C05440=1057.096,54.680,-74.753,171.430,30.537,155.701
C05441=1057.102,54.929,-74.770,171.432,30.540,155.701
C05442=1057.108,55.179,-74.788,171.434,30.542,155.702
C05443=1057.114,55.428,-74.804,171.435,30.544,155.702
C05444=1057.121,55.677,-74.821,171.437,30.547,155.703
C05445=1057.126,55.927,-74.838,171.438,30.549,155.703
C05446=1057.133,56.176,-74.855,171.439,30.552,155.703
C05447=1057.139,56.426,-74.873,171.441,30.554,155.704
C05448=1057.145,56.675,-74.889,171.443,30.557,155.704
C05449=1057.152,56.924,-74.907,171.445,30.559,155.704
C05450=1057.157,57.173,-74.924,171.445,30.561,155.705
C05451=1057.163,57.422,-74.941,171.447,30.563,155.705
C05452=1057.170,57.672,-74.958,171.449,30.566,155.705
C05453=1057.175,57.921,-74.975,171.451,30.568,155.706
C05454=1057.182,58.171,-74.993,171.452,30.571,155.706
C05455=1057.187,58.420,-75.009,171.453,30.573,155.706
C05456=1057.194,58.670,-75.027,171.455,30.576,155.707
C05457=1057.201,58.918,-75.044,171.456,30.578,155.707
C05458=1057.207,59.168,-75.062,171.458,30.580,155.708
C05459=1057.213,59.418,-75.078,171.460,30.583,155.708
C05460=1057.219,59.667,-75.096,171.461,30.585,155.708
C05461=1057.225,59.916,-75.113,171.462,30.588,155.709
C05462=1057.232,60.165,-75.130,171.464,30.590,155.709
C05463=1057.237,60.415,-75.147,171.466,30.593,155.709
C05464=1057.243,60.664,-75.164,171.467,30.594,155.710
C05465=1057.249,60.914,-75.182,171.468,30.597,155.710
C05466=1057.256,61.162,-75.199,171.470,30.599,155.710
C05467=1057.263,61.412,-75.216,171.472,30.602,155.711
C05468=1057.269,61.697,-75.236,171.474,30.605,155.711
C05469=1057.277,61.982,-75.256,171.476,30.607,155.712
C05470=1057.283,62.267,-75.276,171.477,30.610,155.712
C05471=1057.291,62.551,-75.295,171.479,30.613,155.712
C05472=1057.297,62.801,-75.313,171.480,30.615,155.713
C05473=1057.303,63.051,-75.329,171.482,30.618,155.713
C05474=1057.309,63.300,-75.347,171.484,30.620,155.713
C05475=1057.316,63.550,-75.365,171.485,30.622,155.714
C05476=1057.321,63.799,-75.382,171.486,30.624,155.714
C05477=1057.328,64.048,-75.400,171.488,30.627,155.714
C05478=1057.334,64.297,-75.417,171.490,30.629,155.715
C05479=1057.341,64.547,-75.435,171.491,30.632,155.715
C05480=1057.346,64.796,-75.452,171.493,30.634,155.715
C05481=1057.352,65.045,-75.470,171.494,30.636,155.716
C05482=1057.358,65.294,-75.487,171.496,30.639,155.716
C05483=1057.365,65.544,-75.505,171.497,30.641,155.717
C05484=1057.370,65.793,-75.522,171.499,30.644,155.717
C05485=1057.377,66.042,-75.540,171.500,30.647,155.717
C05486=1057.382,66.291,-75.557,171.501,30.649,155.718
C05487=1057.389,66.541,-75.575,171.503,30.651,155.718
C05488=1057.395,66.790,-75.592,171.505,30.653,155.718
C05489=1057.401,67.040,-75.610,171.507,30.656,155.719
C05490=1057.406,67.289,-75.628,171.508,30.659,155.719
C05491=1057.413,67.538,-75.645,171.509,30.661,155.720
C05492=1057.419,67.788,-75.663,171.511,30.663,155.720
C05493=1057.425,68.037,-75.681,171.512,30.666,155.720
C05494=1057.431,68.287,-75.699,171.514,30.668,155.721
C05495=1057.437,68.535,-75.716,171.516,30.671,155.721
C05496=1057.443,68.785,-75.733,171.517,30.673,155.721
C05497=1057.449,69.034,-75.751,171.518,30.675,155.722
C05498=1057.455,69.284,-75.769,171.520,30.678,155.722
C05499=1057.461,69.533,-75.786,171.522,30.680,155.722
C05500=1057.467,69.782,-75.804,171.524,30.683,155.723
C05501=1057.474,70.031,-75.823,171.524,30.685,155.723
C05502=1057.479,70.280,-75.840,171.526,30.688,155.724
C05503=1057.486,70.530,-75.858,171.528,30.690,155.724
C05504=1057.492,70.779,-75.875,171.529,30.693,155.724
C05505=1057.498,71.029,-75.893,171.531,30.695,155.725
C05506=1057.503,71.278,-75.911,171.532,30.698,155.725
C05507=1057.510,71.527,-75.928,171.534,30.700,155.726
C05508=1057.516,71.777,-75.947,171.535,30.702,155.726
C05509=1057.522,72.026,-75.965,171.537,30.705,155.726
C05510=1057.528,72.275,-75.982,171.539,30.708,155.727
C05511=1057.534,72.524,-76.000,171.540,30.710,155.727
C05512=1057.540,72.774,-76.017,171.541,30.712,155.727
C05513=1057.546,73.023,-76.036,171.543,30.715,155.728
C05514=1057.552,73.272,-76.054,171.545,30.717,155.728
C05515=1057.558,73.522,-76.072,171.546,30.720,155.728
C05516=1057.564,73.771,-76.089,171.548,30.722,155.729
C05517=1057.570,74.020,-76.108,171.549,30.725,155.729
C05518=1057.576,74.270,-76.126,171.550,30.727,155.730
C05519=1057.582,74.519,-76.143,171.552,30.730,155.730
C05520=1057.589,74.768,-76.161,171.554,30.732,155.730
C05521=1057.594,75.017,-76.179,171.556,30.735,155.731
C05522=1057.600,75.266,-76.197,171.556,30.737,155.731
C05523=1057.607,75.516,-76.215,171.558,30.739,155.731
C05524=1057.612,75.764,-76.233,171.560,30.742,155.732
C05525=1057.619,76.014,-76.251,171.561,30.744,155.732
C05526=1057.625,76.264,-76.269,171.563,30.747,155.733
C05527=1057.630,76.512,-76.287,171.564,30.749,155.733
C05528=1057.637,76.762,-76.305,171.566,30.752,155.733
C05529=1057.643,77.012,-76.323,171.567,30.754,155.734
C05530=1057.649,77.260,-76.341,171.569,30.757,155.734
C05531=1057.655,77.510,-76.359,171.571,30.759,155.734
C05532=1057.662,77.795,-76.380,171.572,30.762,155.735
C05533=1057.669,78.080,-76.400,171.574,30.765,155.735
C05534=1057.676,78.364,-76.421,171.576,30.767,155.736
C05535=1057.683,78.649,-76.442,171.578,30.771,155.736
C05536=1057.689,78.899,-76.460,171.579,30.773,155.737
C05537=1057.695,79.147,-76.478,171.580,30.775,155.737
C05538=1057.700,79.397,-76.497,171.582,30.778,155.737
C05539=1057.706,79.647,-76.515,171.584,30.781,155.738
C05540=1057.712,79.896,-76.533,171.585,30.783,155.738
C05541=1057.718,80.145,-76.551,171.587,30.785,155.738
C05542=1057.725,80.394,-76.570,171.588,30.788,155.739
C05543=1057.730,80.643,-76.587,171.589,30.791,155.739
C05544=1057.736,80.893,-76.606,171.591,30.793,155.740
C05545=1057.742,81.143,-76.624,171.593,30.795,155.740
C05546=1057.748,81.391,-76.643,171.595,30.798,155.740
C05547=1057.754,81.641,-76.661,171.596,30.801,155.741
C05548=1057.760,81.890,-76.679,171.597,30.803,155.741
C05549=1057.766,82.139,-76.697,171.599,30.805,155.742
C05550=1057.772,82.388,-76.716,171.601,30.808,155.742
C05551=1057.778,82.638,-76.735,171.602,30.811,155.742
C05552=1057.784,82.887,-76.753,171.604,30.813,155.743
C05553=1057.790,83.136,-76.771,171.605,30.815,155.743
C05554=1057.796,83.385,-76.789,171.606,30.818,155.744
C05555=1057.802,83.635,-76.807,171.608,30.821,155.744
C05556=1057.808,83.885,-76.826,171.610,30.823,155.744
C05557=1057.814,84.133,-76.844,171.612,30.825,155.745
C05558=1057.820,84.382,-76.863,171.613,30.828,155.745
C05559=1057.826,84.632,-76.881,171.614,30.830,155.745
C05560=1057.833,84.881,-76.899,171.616,30.833,155.746
C05561=1057.837,85.130,-76.918,171.618,30.835,155.746
C05562=1057.844,85.379,-76.936,171.619,30.838,155.747
C05563=1057.850,85.629,-76.955,171.621,30.840,155.747
C05564=1057.856,85.878,-76.973,171.622,30.843,155.747
C05565=1057.862,86.127,-76.991,171.623,30.845,155.748
C05566=1057.868,86.376,-77.010,171.625,30.847,155.748
C05567=1057.874,86.626,-77.028,171.627,30.850,155.748
C05568=1057.880,86.875,-77.047,171.629,30.853,155.749
C05569=1057.887,87.124,-77.066,171.630,30.855,155.749
C05570=1057.892,87.373,-77.083,171.631,30.857,155.750
C05571=1057.898,87.623,-77.102,171.633,30.860,155.750
C05572=1057.905,87.872,-77.121,171.635,30.863,155.750
C05573=1057.911,88.121,-77.140,171.636,30.865,155.751
C05574=1057.917,88.371,-77.158,171.638,30.867,155.751
C05575=1057.923,88.619,-77.176,171.639,30.870,155.752
C05576=1057.929,88.868,-77.195,171.641,30.872,155.752
C05577=1057.935,89.118,-77.214,171.642,30.875,155.752
C05578=1057.941,89.367,-77.232,171.644,30.877,155.753
C05579=1057.948,89.616,-77.250,171.646,30.880,155.753
C05580=1057.953,89.866,-77.270,171.648,30.882,155.753
C05581=1057.960,90.115,-77.288,171.648,30.885,155.754
C05582=1057.965,90.364,-77.306,171.650,30.887,155.754
C05583=1057.972,90.613,-77.325,171.652,30.890,155.754
C05584=1057.977,90.863,-77.344,171.654,30.892,155.755
C05585=1057.984,91.112,-77.362,171.655,30.895,155.755
C05586=1057.989,91.361,-77.382,171.656,30.897,155.756
C05587=1057.996,91.610,-77.400,171.658,30.900,155.756
C05588=1058.001,91.860,-77.418,171.659,30.902,155.756
C05589=1058.007,92.109,-77.437,171.661,30.905,155.757
C05590=1058.013,92.358,-77.456,171.663,30.907,155.757
C05591=1058.019,92.607,-77.475,171.665,30.910,155.758
C05592=1058.025,92.857,-77.494,171.665,30.912,155.758
C05593=1058.031,93.106,-77.513,171.667,30.915,155.758
C05594=1058.036,93.355,-77.532,171.669,30.917,155.759
C05595=1058.043,93.604,-77.550,171.671,30.920,155.759
C05596=1058.049,93.889,-77.572,171.673,30.923,155.760
C05597=1058.057,94.174,-77.593,171.674,30.926,155.760
C05598=1058.063,94.458,-77.615,171.676,30.929,155.761
C05599=1058.070,94.743,-77.637,171.678,30.931,155.761
C05600=1058.076,94.992,-77.655,171.679,30.934,155.761
C05601=1058.082,95.242,-77.675,171.681,30.937,155.762
C05602=1058.089,95.491,-77.693,171.682,30.939,155.762
C05603=1058.094,95.740,-77.712,171.684,30.941,155.763
C05604=1058.101,95.990,-77.731,171.685,30.944,155.763
C05605=1058.106,96.239,-77.750,171.687,30.947,155.763
C05606=1058.112,96.487,-77.769,171.689,30.949,155.764
C05607=1058.118,96.737,-77.788,171.691,30.951,155.764
C05608=1058.124,96.986,-77.806,171.691,30.954,155.764
C05609=1058.130,97.235,-77.826,171.693,30.957,155.765
C05610=1058.136,97.484,-77.844,171.695,30.959,155.765
C05611=1058.142,97.734,-77.864,171.697,30.961,155.766
C05612=1058.148,97.983,-77.883,171.698,30.964,155.766
C05613=1058.154,98.232,-77.902,171.700,30.967,155.766
C05614=1058.160,98.482,-77.921,171.701,30.969,155.767
C05615=1058.166,98.731,-77.939,171.703,30.971,155.767
C05616=1058.172,98.980,-77.959,171.704,30.974,155.768
C05617=1058.178,99.230,-77.977,171.706,30.977,155.768
C05618=1058.184,99.478,-77.997,171.708,30.979,155.768
C05619=1058.191,99.728,-78.016,171.710,30.981,155.769
C05620=1058.197,99.977,-78.035,171.710,30.984,155.769
C05621=1058.203,100.226,-78.054,171.712,30.987,155.770
C05622=1058.209,100.476,-78.073,171.714,30.989,155.770
C05623=1058.215,100.725,-78.092,171.716,30.991,155.770
C05624=1058.221,100.974,-78.111,171.718,30.994,155.771
C05625=1058.227,101.223,-78.131,171.718,30.997,155.771
C05626=1058.232,101.472,-78.150,171.720,30.999,155.772
C05627=1058.239,101.721,-78.169,171.722,31.002,155.772
C05628=1058.245,101.971,-78.188,171.724,31.004,155.772
C05629=1058.250,102.220,-78.207,171.725,31.006,155.773
C05630=1058.256,102.468,-78.227,171.727,31.009,155.773
C05631=1058.262,102.718,-78.246,171.728,31.012,155.773
C05632=1058.268,102.967,-78.265,171.730,31.015,155.774
C05633=1058.273,103.216,-78.284,171.731,31.017,155.774
C05634=1058.279,103.465,-78.304,171.733,31.019,155.775
C05635=1058.285,103.715,-78.323,171.735,31.022,155.775
C05636=1058.292,103.964,-78.342,171.737,31.024,155.775
C05637=1058.298,104.213,-78.362,171.737,31.027,155.776
C05638=1058.303,104.462,-78.381,171.739,31.030,155.776
C05639=1058.309,104.711,-78.400,171.741,31.032,155.777
C05640=1058.315,104.961,-78.419,171.743,31.034,155.777
C05641=1058.321,105.209,-78.439,171.744,31.037,155.777
C05642=1058.327,105.459,-78.458,171.746,31.040,155.778
C05643=1058.333,105.708,-78.477,171.747,31.042,155.778
C05644=1058.339,105.957,-78.497,171.749,31.045,155.779
C05645=1058.345,106.206,-78.516,171.751,31.048,155.779
C05646=1058.351,106.456,-78.535,171.752,31.050,155.779
C05647=1058.357,106.704,-78.555,171.754,31.052,155.780
C05648=1058.363,106.955,-78.575,171.756,31.055,155.780
C05649=1058.369,107.203,-78.595,171.757,31.058,155.781
C05650=1058.376,107.452,-78.613,171.758,31.060,155.781
C05651=1058.381,107.702,-78.633,171.760,31.062,155.781
C05652=1058.387,107.951,-78.653,171.762,31.065,155.782
C05653=1058.393,108.200,-78.672,171.764,31.068,155.782
C05654=1058.399,108.449,-78.692,171.765,31.070,155.783
C05655=1058.405,108.698,-78.711,171.766,31.073,155.783
C05656=1058.411,108.947,-78.730,171.768,31.075,155.783
C05657=1058.417,109.196,-78.750,171.770,31.077,155.784
C05658=1058.423,109.446,-78.769,171.772,31.080,155.784
C05659=1058.429,109.695,-78.789,171.773,31.083,155.785
C05660=1058.436,109.980,-78.811,171.775,31.085,155.785
C05661=1058.443,110.264,-78.834,171.777,31.088,155.785
C05662=1058.450,110.550,-78.856,171.779,31.091,155.786
C05663=1058.457,110.835,-78.878,171.781,31.094,155.786
C05664=1058.463,111.083,-78.898,171.782,31.097,155.787
C05665=1058.469,111.333,-78.917,171.784,31.099,155.787
C05666=1058.475,111.582,-78.937,171.785,31.102,155.788
C05667=1058.481,111.830,-78.957,171.787,31.104,155.788
C05668=1058.486,112.080,-78.976,171.789,31.107,155.788
C05669=1058.492,112.329,-78.996,171.790,31.109,155.789
C05670=1058.498,112.578,-79.015,171.792,31.112,155.789
C05671=1058.505,112.828,-79.036,171.794,31.115,155.790
C05672=1058.510,113.077,-79.055,171.795,31.117,155.790
C05673=1058.516,113.326,-79.075,171.797,31.119,155.790
C05674=1058.522,113.575,-79.095,171.798,31.122,155.791
C05675=1058.528,113.824,-79.114,171.800,31.124,155.791
C05676=1058.534,114.073,-79.134,171.802,31.127,155.791
C05677=1058.540,114.322,-79.154,171.804,31.130,155.792
C05678=1058.546,114.571,-79.173,171.805,31.132,155.792
C05679=1058.551,114.821,-79.194,171.806,31.135,155.793
C05680=1058.557,115.070,-79.214,171.808,31.138,155.793
C05681=1058.563,115.319,-79.233,171.810,31.140,155.794
C05682=1058.569,115.568,-79.253,171.812,31.143,155.794
C05683=1058.575,115.817,-79.273,171.814,31.146,155.794
C05684=1058.580,116.067,-79.293,171.814,31.148,155.795
C05685=1058.586,116.315,-79.313,171.816,31.151,155.795
C05686=1058.592,116.564,-79.333,171.818,31.153,155.796
C05687=1058.598,116.813,-79.353,171.820,31.156,155.796
C05688=1058.604,117.064,-79.373,171.822,31.158,155.796
C05689=1058.610,117.312,-79.393,171.823,31.161,155.797
C05690=1058.616,117.561,-79.413,171.824,31.163,155.797
C05691=1058.622,117.810,-79.433,171.826,31.166,155.798
C05692=1058.627,118.059,-79.452,171.828,31.169,155.798
C05693=1058.633,118.309,-79.473,171.830,31.171,155.798
C05694=1058.639,118.558,-79.493,171.831,31.174,155.799
C05695=1058.645,118.807,-79.513,171.833,31.177,155.799
C05696=1058.651,119.056,-79.533,171.834,31.179,155.800
C05697=1058.656,119.305,-79.553,171.836,31.182,155.800
C05698=1058.662,119.554,-79.573,171.838,31.185,155.801
C05699=1058.668,119.803,-79.593,171.839,31.187,155.801
C05700=1058.675,120.053,-79.613,171.841,31.190,155.801
C05701=1058.680,120.302,-79.634,171.843,31.192,155.802
C05702=1058.686,120.551,-79.654,171.844,31.194,155.802
C05703=1058.692,120.799,-79.674,171.846,31.197,155.803
C05704=1058.698,121.049,-79.693,171.847,31.200,155.803
C05705=1058.703,121.299,-79.714,171.849,31.202,155.803
C05706=1058.709,121.547,-79.734,171.851,31.205,155.804
C05707=1058.715,121.796,-79.754,171.853,31.208,155.804
C05708=1058.721,122.045,-79.774,171.854,31.210,155.805
C05709=1058.727,122.295,-79.795,171.856,31.213,155.805
C05710=1058.733,122.544,-79.815,171.857,31.215,155.805
C05711=1058.739,122.792,-79.835,171.859,31.218,155.806
C05712=1058.745,123.042,-79.855,171.861,31.220,155.806
C05713=1058.751,123.291,-79.876,171.863,31.223,155.807
C05714=1058.757,123.540,-79.895,171.865,31.225,155.807
C05715=1058.763,123.789,-79.915,171.866,31.228,155.807
C05716=1058.769,124.039,-79.936,171.867,31.231,155.808
C05717=1058.775,124.287,-79.956,171.869,31.233,155.808
C05718=1058.781,124.536,-79.976,171.871,31.236,155.809
C05719=1058.786,124.785,-79.997,171.873,31.239,155.809
C05720=1058.793,125.035,-80.017,171.875,31.241,155.810
C05721=1058.799,125.284,-80.037,171.876,31.243,155.810
C05722=1058.804,125.533,-80.058,171.877,31.246,155.810
C05723=1058.811,125.782,-80.078,171.879,31.248,155.811
C05724=1058.817,126.067,-80.101,171.881,31.252,155.811
C05725=1058.824,126.351,-80.124,171.884,31.255,155.812
C05726=1058.831,126.636,-80.147,171.886,31.257,155.812
C05727=1058.838,126.921,-80.171,171.887,31.260,155.813
C05728=1058.844,127.170,-80.191,171.889,31.263,155.813
C05729=1058.850,127.419,-80.211,171.890,31.266,155.813
C05730=1058.855,127.669,-80.232,171.892,31.268,155.814
C05731=1058.862,127.917,-80.252,171.894,31.270,155.814
C05732=1058.868,128.167,-80.273,171.896,31.273,155.815
C05733=1058.874,128.415,-80.293,171.897,31.276,155.815
C05734=1058.880,128.664,-80.313,171.899,31.278,155.815
C05735=1058.886,128.914,-80.334,171.901,31.281,155.816
C05736=1058.891,129.163,-80.354,171.903,31.284,155.816
C05737=1058.897,129.412,-80.374,171.904,31.285,155.817
C05738=1058.904,129.661,-80.395,171.906,31.288,155.817
C05739=1058.910,129.910,-80.416,171.908,31.291,155.817
C05740=1058.916,130.159,-80.436,171.909,31.293,155.818
C05741=1058.922,130.408,-80.456,171.911,31.296,155.818
C05742=1058.928,130.658,-80.477,171.913,31.299,155.819
C05743=1058.934,130.906,-80.498,171.915,31.301,155.819
C05744=1058.940,131.155,-80.518,171.917,31.303,155.819
C05745=1058.946,131.405,-80.538,171.918,31.306,155.820
C05746=1058.952,131.654,-80.558,171.920,31.309,155.820
C05747=1058.958,131.903,-80.580,171.921,31.311,155.821
C05748=1058.964,132.152,-80.600,171.923,31.314,155.821
C05749=1058.970,132.401,-80.621,171.925,31.317,155.821
C05750=1058.976,132.650,-80.641,171.927,31.319,155.822
C05751=1058.982,132.899,-80.662,171.929,31.322,155.822
C05752=1058.988,133.149,-80.683,171.930,31.324,155.823
C05753=1058.994,133.398,-80.703,171.931,31.327,155.823
C05754=1058.999,133.646,-80.724,171.933,31.330,155.824
C05755=1059.005,133.896,-80.745,171.935,31.332,155.824
C05756=1059.011,134.144,-80.766,171.937,31.335,155.824
C05757=1059.017,134.394,-80.787,171.939,31.338,155.825
C05758=1059.023,134.643,-80.807,171.941,31.340,155.825
C05759=1059.029,134.891,-80.828,171.943,31.343,155.826
C05760=1059.035,135.141,-80.849,171.944,31.346,155.826
C05761=1059.041,135.390,-80.869,171.945,31.348,155.826
C05762=1059.047,135.639,-80.891,171.947,31.351,155.827
C05763=1059.052,135.888,-80.911,171.949,31.353,155.827
C05764=1059.059,136.137,-80.932,171.951,31.356,155.828
C05765=1059.064,136.386,-80.953,171.953,31.358,155.828
C05766=1059.070,136.635,-80.974,171.954,31.361,155.828
C05767=1059.076,136.884,-80.994,171.956,31.363,155.829
C05768=1059.082,137.133,-81.016,171.958,31.366,155.829
C05769=1059.088,137.382,-81.036,171.960,31.369,155.830
C05770=1059.094,137.631,-81.057,171.961,31.371,155.830
C05771=1059.100,137.881,-81.078,171.963,31.374,155.831
C05772=1059.105,138.129,-81.099,171.965,31.376,155.831
C05773=1059.112,138.379,-81.120,171.966,31.379,155.831
C05774=1059.118,138.627,-81.141,171.968,31.382,155.832
C05775=1059.123,138.877,-81.162,171.970,31.384,155.832
C05776=1059.129,139.125,-81.183,171.972,31.387,155.833
C05777=1059.136,139.375,-81.203,171.974,31.390,155.833
C05778=1059.141,139.623,-81.225,171.976,31.392,155.833
C05779=1059.147,139.873,-81.246,171.978,31.395,155.834
C05780=1059.153,140.121,-81.266,171.979,31.398,155.834
C05781=1059.160,140.371,-81.288,171.980,31.400,155.835
C05782=1059.165,140.620,-81.309,171.982,31.403,155.835
C05783=1059.171,140.869,-81.330,171.984,31.405,155.836
C05784=1059.176,141.118,-81.351,171.986,31.408,155.836
C05785=1059.182,141.367,-81.372,171.988,31.411,155.836
C05786=1059.188,141.616,-81.394,171.990,31.413,155.837
C05787=1059.194,141.866,-81.415,171.991,31.416,155.837
C05788=1059.200,142.150,-81.439,171.993,31.419,155.838
C05789=1059.208,142.434,-81.463,171.995,31.422,155.838
C05790=1059.215,142.719,-81.487,171.997,31.425,155.839
C05791=1059.221,143.004,-81.511,172.000,31.428,155.839
C05792=1059.226,143.253,-81.532,172.002,31.431,155.840
C05793=1059.233,143.502,-81.554,172.003,31.434,155.840
C05794=1059.239,143.750,-81.575,172.004,31.436,155.841
C05795=1059.245,144.000,-81.596,172.006,31.439,155.841
C05796=1059.250,144.248,-81.617,172.008,31.441,155.841
C05797=1059.256,144.498,-81.639,172.010,31.444,155.842
C05798=1059.262,144.746,-81.660,172.012,31.447,155.842
C05799=1059.268,144.996,-81.681,172.014,31.449,155.843
C05800=1059.274,145.233,-81.702,172.015,31.452,155.843
C05801=1059.279,145.470,-81.721,172.017,31.455,155.843
C05802=1059.285,145.707,-81.742,172.019,31.457,155.844
C05803=1059.290,145.944,-81.762,172.021,31.459,155.844
C05804=1059.296,146.181,-81.783,172.022,31.462,155.845
C05805=1059.302,146.418,-81.802,172.024,31.464,155.845
C05806=1059.308,146.655,-81.823,172.026,31.467,155.845
C05807=1059.313,146.892,-81.843,172.027,31.470,155.846
C05808=1059.319,147.141,-81.865,172.029,31.472,155.846
C05809=1059.325,147.391,-81.886,172.031,31.475,155.847
C05810=1059.331,147.639,-81.907,172.033,31.478,155.847
C05811=1059.337,147.888,-81.929,172.035,31.480,155.848
C05812=1059.342,148.137,-81.950,172.037,31.483,155.848
C05813=1059.348,148.386,-81.972,172.039,31.485,155.848
C05814=1059.355,148.635,-81.994,172.040,31.488,155.849
C05815=1059.360,148.884,-82.015,172.042,31.491,155.849
C05816=1059.366,149.134,-82.036,172.044,31.493,155.850
C05817=1059.372,149.382,-82.057,172.045,31.496,155.850
C05818=1059.378,149.631,-82.079,172.047,31.498,155.851
C05819=1059.384,149.881,-82.100,172.049,31.501,155.851
C05820=1059.390,150.129,-82.122,172.051,31.504,155.851
C05821=1059.396,150.378,-82.143,172.052,31.506,155.852
C05822=1059.401,150.628,-82.166,172.054,31.510,155.852
C05823=1059.407,150.876,-82.187,172.056,31.512,155.853
C05824=1059.413,151.125,-82.208,172.058,31.515,155.853
C05825=1059.419,151.375,-82.230,172.060,31.517,155.854
C05826=1059.425,151.623,-82.251,172.062,31.520,155.854
C05827=1059.431,151.872,-82.273,172.064,31.523,155.854
C05828=1059.436,152.122,-82.295,172.065,31.525,155.855
C05829=1059.442,152.370,-82.317,172.067,31.528,155.855
C05830=1059.448,152.619,-82.339,172.069,31.531,155.856
C05831=1059.454,152.868,-82.360,172.071,31.533,155.856
C05832=1059.460,153.117,-82.382,172.073,31.536,155.857
C05833=1059.466,153.366,-82.403,172.075,31.539,155.857
C05834=1059.471,153.615,-82.426,172.077,31.542,155.857
C05835=1059.477,153.864,-82.447,172.078,31.544,155.858
C05836=1059.483,154.113,-82.468,172.080,31.547,155.858
C05837=1059.489,154.362,-82.490,172.082,31.550,155.859
C05838=1059.496,154.612,-82.512,172.084,31.552,155.859
C05839=1059.501,154.860,-82.534,172.086,31.555,155.860
C05840=1059.507,155.109,-82.556,172.088,31.558,155.860
C05841=1059.513,155.358,-82.578,172.090,31.560,155.860
C05842=1059.519,155.607,-82.599,172.092,31.563,155.861
C05843=1059.524,155.856,-82.621,172.093,31.566,155.861
C05844=1059.530,156.105,-82.643,172.095,31.569,155.862
C05845=1059.537,156.354,-82.665,172.097,31.571,155.862
C05846=1059.541,156.603,-82.687,172.099,31.574,155.863
C05847=1059.548,156.852,-82.709,172.101,31.576,155.863
C05848=1059.554,157.101,-82.730,172.103,31.580,155.864
C05849=1059.560,157.350,-82.753,172.105,31.582,155.864
C05850=1059.565,157.599,-82.774,172.106,31.585,155.864
C05851=1059.571,157.848,-82.796,172.108,31.588,155.865
C05852=1059.579,158.156,-82.824,172.111,31.591,155.865
C05853=1059.586,158.464,-82.851,172.113,31.594,155.866
C05854=1059.593,158.772,-82.877,172.116,31.597,155.866
C05855=1059.600,159.081,-82.905,172.118,31.601,155.867
C05856=1059.606,159.330,-82.927,172.119,31.604,155.868
C05857=1059.613,159.579,-82.949,172.121,31.607,155.868
C05858=1059.617,159.828,-82.971,172.123,31.609,155.868
C05859=1059.624,160.076,-82.993,172.125,31.612,155.869
C05860=1059.630,160.325,-83.015,172.127,31.614,155.869
C05861=1059.636,160.574,-83.038,172.129,31.617,155.870
C05862=1059.642,160.824,-83.060,172.131,31.620,155.870
C05863=1059.647,161.073,-83.082,172.133,31.623,155.871
C05864=1059.653,161.321,-83.104,172.134,31.625,155.871
C05865=1059.659,161.570,-83.126,172.136,31.628,155.871
C05866=1059.664,161.819,-83.149,172.138,31.631,155.872
C05867=1059.670,162.068,-83.170,172.140,31.634,155.872
C05868=1059.676,162.317,-83.193,172.142,31.637,155.873
C05869=1059.681,162.566,-83.215,172.144,31.640,155.873
C05870=1059.688,162.815,-83.238,172.146,31.642,155.874
C05871=1059.693,163.064,-83.260,172.147,31.645,155.874
C05872=1059.698,163.313,-83.283,172.150,31.648,155.875
C05873=1059.704,163.562,-83.304,172.152,31.651,155.875
C05874=1059.710,163.811,-83.327,172.154,31.654,155.876
C05875=1059.715,164.060,-83.349,172.156,31.657,155.876
C05876=1059.721,164.308,-83.372,172.158,31.659,155.877
C05877=1059.727,164.557,-83.394,172.160,31.662,155.877
C05878=1059.732,164.806,-83.416,172.162,31.665,155.877
C05879=1059.738,165.055,-83.439,172.163,31.668,155.878
C05880=1059.744,165.305,-83.461,172.165,31.670,155.878
C05881=1059.750,165.553,-83.484,172.167,31.674,155.879
C05882=1059.755,165.802,-83.507,172.169,31.676,155.879
C05883=1059.761,166.051,-83.529,172.171,31.679,155.880
C05884=1059.767,166.300,-83.551,172.173,31.682,155.880
C05885=1059.773,166.549,-83.573,172.175,31.685,155.881
C05886=1059.778,166.798,-83.596,172.176,31.687,155.881
C05887=1059.785,167.047,-83.619,172.178,31.690,155.882
C05888=1059.790,167.296,-83.641,172.180,31.693,155.882
C05889=1059.795,167.544,-83.664,172.182,31.696,155.883
C05890=1059.801,167.793,-83.686,172.184,31.699,155.883
C05891=1059.808,168.042,-83.709,172.187,31.702,155.883
C05892=1059.813,168.291,-83.731,172.189,31.704,155.884
C05893=1059.819,168.540,-83.754,172.191,31.707,155.884
C05894=1059.824,168.789,-83.777,172.192,31.710,155.885
C05895=1059.831,169.038,-83.799,172.194,31.713,155.885
C05896=1059.836,169.287,-83.822,172.196,31.716,155.886
C05897=1059.841,169.536,-83.844,172.198,31.719,155.886
C05898=1059.847,169.784,-83.867,172.200,31.721,155.887
C05899=1059.853,170.033,-83.890,172.202,31.724,155.887
C05900=1059.859,170.283,-83.912,172.204,31.727,155.888
C05901=1059.865,170.531,-83.935,172.206,31.730,155.888
C05902=1059.871,170.780,-83.958,172.207,31.733,155.889
C05903=1059.876,171.029,-83.980,172.210,31.735,155.889
C05904=1059.883,171.278,-84.003,172.212,31.738,155.889
C05905=1059.888,171.527,-84.026,172.214,31.741,155.890
C05906=1059.894,171.776,-84.048,172.216,31.744,155.890
C05907=1059.900,172.025,-84.071,172.218,31.747,155.891
C05908=1059.905,172.274,-84.094,172.220,31.750,155.891
C05909=1059.912,172.523,-84.116,172.222,31.752,155.892
C05910=1059.918,172.772,-84.139,172.223,31.755,155.892
C05911=1059.923,173.020,-84.162,172.225,31.758,155.893
C05912=1059.929,173.269,-84.185,172.228,31.761,155.893
C05913=1059.935,173.518,-84.208,172.230,31.763,155.894
C05914=1059.941,173.767,-84.230,172.232,31.767,155.894
C05915=1059.947,174.016,-84.253,172.234,31.769,155.895
C05916=1059.954,174.300,-84.279,172.236,31.772,155.895
C05917=1059.960,174.584,-84.306,172.238,31.776,155.896
C05918=1059.967,174.868,-84.331,172.240,31.779,155.896
C05919=1059.973,175.151,-84.357,172.243,31.782,155.897
C05920=1059.979,175.401,-84.381,172.245,31.785,155.897
C05921=1059.985,175.650,-84.404,172.247,31.788,155.898
C05922=1059.992,175.898,-84.426,172.249,31.791,155.898
C05923=1059.997,176.147,-84.449,172.251,31.793,155.898
C05924=1060.003,176.396,-84.472,172.253,31.796,155.899
C05925=1060.009,176.645,-84.495,172.255,31.799,155.899
C05926=1060.015,176.894,-84.518,172.257,31.802,155.900
C05927=1060.020,177.143,-84.541,172.259,31.804,155.900
C05928=1060.027,177.391,-84.563,172.261,31.808,155.901
C05929=1060.033,177.640,-84.586,172.263,31.810,155.901
C05930=1060.038,177.889,-84.609,172.265,31.813,155.902
C05931=1060.045,178.139,-84.632,172.268,31.816,155.902
C05932=1060.050,178.388,-84.655,172.270,31.819,155.903
C05933=1060.056,178.636,-84.679,172.271,31.821,155.903
C05934=1060.062,178.885,-84.702,172.273,31.825,155.904
C05935=1060.069,179.133,-84.724,172.275,31.827,155.904
C05936=1060.074,179.382,-84.747,172.277,31.830,155.904
C05937=1060.080,179.631,-84.770,172.280,31.833,155.905
C05938=1060.086,179.881,-84.793,172.282,31.836,155.905
C05939=1060.092,180.130,-84.816,172.284,31.838,155.906
C05940=1060.098,180.378,-84.840,172.286,31.841,155.906
C05941=1060.104,180.627,-84.863,172.288,31.844,155.907
C05942=1060.110,180.876,-84.886,172.290,31.847,155.907
C05943=1060.115,181.125,-84.909,172.292,31.850,155.908
C05944=1060.123,181.373,-84.932,172.294,31.853,155.908
C05945=1060.128,181.622,-84.955,172.296,31.855,155.909
C05946=1060.134,181.871,-84.978,172.298,31.858,155.909
C05947=1060.140,182.120,-85.001,172.301,31.861,155.910
C05948=1060.146,182.368,-85.025,172.303,31.864,155.910
C05949=1060.152,182.618,-85.048,172.305,31.867,155.911
C05950=1060.158,182.867,-85.071,172.306,31.869,155.911
C05951=1060.164,183.116,-85.094,172.308,31.872,155.911
C05952=1060.170,183.364,-85.118,172.311,31.875,155.912
C05953=1060.176,183.614,-85.141,172.313,31.878,155.912
C05954=1060.183,183.862,-85.163,172.315,31.881,155.913
C05955=1060.189,184.110,-85.187,172.317,31.884,155.913
C05956=1060.194,184.359,-85.210,172.320,31.886,155.914
C05957=1060.200,184.609,-85.234,172.322,31.890,155.914
C05958=1060.206,184.857,-85.257,172.324,31.892,155.915
C05959=1060.212,185.106,-85.280,172.325,31.895,155.915
C05960=1060.217,185.355,-85.305,172.327,31.898,155.916
C05961=1060.223,185.604,-85.328,172.330,31.901,155.916
C05962=1060.229,185.852,-85.351,172.332,31.905,155.917
C05963=1060.234,186.102,-85.375,172.334,31.907,155.917
C05964=1060.240,186.350,-85.399,172.336,31.910,155.918
C05965=1060.245,186.600,-85.422,172.338,31.913,155.918
C05966=1060.251,186.848,-85.446,172.341,31.916,155.919
C05967=1060.257,187.097,-85.469,172.342,31.919,155.919
C05968=1060.262,187.345,-85.493,172.344,31.923,155.920
C05969=1060.269,187.594,-85.517,172.346,31.925,155.920
C05970=1060.274,187.843,-85.541,172.348,31.928,155.921
C05971=1060.280,188.092,-85.564,172.351,31.931,155.921
C05972=1060.286,188.341,-85.587,172.353,31.934,155.922
C05973=1060.291,188.589,-85.612,172.355,31.937,155.922
C05974=1060.297,188.839,-85.635,172.357,31.940,155.923
C05975=1060.303,189.087,-85.659,172.360,31.943,155.923
C05976=1060.309,189.336,-85.683,172.361,31.946,155.924
C05977=1060.314,189.585,-85.706,172.363,31.949,155.924
C05978=1060.320,189.834,-85.730,172.365,31.952,155.925
C05979=1060.326,190.082,-85.754,172.368,31.956,155.925
C05980=1060.333,190.366,-85.781,172.370,31.959,155.926
C05981=1060.339,190.649,-85.808,172.373,31.962,155.926
C05982=1060.346,190.933,-85.835,172.375,31.966,155.927
C05983=1060.353,191.216,-85.863,172.378,31.969,155.928
C05984=1060.358,191.465,-85.887,172.379,31.972,155.928
C05985=1060.364,191.714,-85.910,172.381,31.975,155.928
C05986=1060.369,191.962,-85.934,172.384,31.978,155.929
C05987=1060.376,192.211,-85.958,172.386,31.981,155.929
C05988=1060.381,192.460,-85.982,172.388,31.984,155.930
C05989=1060.387,192.709,-86.005,172.390,31.987,155.931
C05990=1060.393,192.958,-86.030,172.393,31.990,155.931
C05991=1060.399,193.207,-86.053,172.395,31.993,155.932
C05992=1060.404,193.455,-86.078,172.397,31.996,155.932
C05993=1060.411,193.705,-86.101,172.399,31.999,155.932
C05994=1060.416,193.953,-86.125,172.401,32.002,155.933
C05995=1060.423,194.202,-86.149,172.403,32.005,155.934
C05996=1060.429,194.451,-86.173,172.405,32.008,155.934
C05997=1060.434,194.699,-86.197,172.408,32.011,155.935
C05998=1060.441,194.948,-86.221,172.410,32.014,155.935
C05999=1060.446,195.197,-86.246,172.412,32.017,155.935
C06000=1060.452,195.446,-86.268,172.415,32.020,155.936
C06001=1060.457,195.695,-86.293,172.417,32.023,155.937
C06002=1060.463,195.943,-86.317,172.418,32.026,155.937
C06003=1060.469,196.192,-86.341,172.421,32.029,155.938
C06004=1060.475,196.441,-86.365,172.423,32.032,155.938
C06005=1060.481,196.689,-86.389,172.425,32.035,155.939
C06006=1060.487,196.938,-86.413,172.428,32.038,155.939
C06007=1060.493,197.187,-86.438,172.430,32.041,155.940
C06008=1060.499,197.436,-86.462,172.432,32.044,155.940
C06009=1060.505,197.684,-86.486,172.435,32.047,155.941
C06010=1060.511,197.933,-86.510,172.437,32.050,155.941
C06011=1060.517,198.182,-86.534,172.439,32.053,155.942
C06012=1060.522,198.431,-86.559,172.441,32.056,155.942
C06013=1060.528,198.680,-86.582,172.443,32.059,155.943
C06014=1060.534,198.929,-86.607,172.445,32.063,155.943
C06015=1060.540,199.177,-86.631,172.448,32.066,155.944
C06016=1060.546,199.426,-86.655,172.450,32.068,155.944
C06017=1060.552,199.675,-86.679,172.452,32.072,155.945
C06018=1060.558,199.924,-86.704,172.455,32.075,155.945
C06019=1060.564,200.172,-86.727,172.457,32.077,155.946
C06020=1060.570,200.421,-86.753,172.459,32.081,155.946
C06021=1060.577,200.669,-86.776,172.461,32.084,155.947
C06022=1060.582,200.919,-86.801,172.463,32.087,155.947
C06023=1060.588,201.167,-86.825,172.465,32.090,155.948
C06024=1060.594,201.416,-86.849,172.468,32.093,155.948
C06025=1060.600,201.665,-86.873,172.470,32.096,155.949
C06026=1060.606,201.914,-86.897,172.472,32.099,155.949
C06027=1060.612,202.162,-86.922,172.475,32.102,155.950
C06028=1060.618,202.411,-86.947,172.477,32.105,155.950
C06029=1060.623,202.659,-86.971,172.480,32.108,155.951
C06030=1060.630,202.908,-86.995,172.482,32.111,155.951
C06031=1060.635,203.156,-87.020,172.483,32.115,155.952
C06032=1060.641,203.406,-87.045,172.486,32.118,155.952
C06033=1060.647,203.654,-87.069,172.488,32.121,155.953
C06034=1060.652,203.904,-87.094,172.490,32.124,155.954
C06035=1060.658,204.152,-87.119,172.493,32.127,155.954
C06036=1060.665,204.401,-87.143,172.495,32.130,155.955
C06037=1060.671,204.650,-87.167,172.498,32.133,155.955
C06038=1060.676,204.898,-87.192,172.500,32.136,155.956
C06039=1060.682,205.147,-87.217,172.502,32.140,155.956
C06040=1060.687,205.396,-87.241,172.505,32.143,155.957
C06041=1060.694,205.644,-87.267,172.506,32.146,155.957
C06042=1060.699,205.893,-87.291,172.508,32.149,155.958
C06043=1060.705,206.142,-87.316,172.511,32.153,155.958
C06044=1060.730,207.190,-87.420,172.690,32.237,155.967
C06045=1060.736,207.419,-87.443,172.692,32.241,155.968
C06046=1060.741,207.648,-87.466,172.694,32.245,155.969
C06047=1060.747,207.877,-87.490,172.696,32.248,155.969
C06048=1060.752,208.106,-87.514,172.696,32.252,155.970
C06049=1060.758,208.335,-87.537,172.698,32.255,155.971
C06050=1060.764,208.564,-87.561,172.700,32.259,155.971
C06051=1060.770,208.793,-87.584,172.702,32.263,155.972
C06052=1060.775,209.022,-87.608,172.704,32.267,155.973
C06053=1060.782,209.270,-87.633,172.706,32.271,155.974
C06054=1060.787,209.519,-87.659,172.708,32.275,155.974
C06055=1060.793,209.767,-87.685,172.710,32.279,155.975
C06056=1060.800,210.016,-87.711,172.712,32.283,155.976
C06057=1060.806,210.265,-87.736,172.714,32.287,155.976
C06058=1060.811,210.514,-87.762,172.716,32.291,155.977
C06059=1060.818,210.762,-87.788,172.717,32.295,155.978
C06060=1060.824,211.011,-87.813,172.719,32.299,155.979
C06061=1060.830,211.260,-87.840,172.721,32.303,155.979
C06062=1060.837,211.508,-87.866,172.723,32.306,155.980
C06063=1060.843,211.757,-87.891,172.725,32.311,155.981
C06064=1060.848,212.006,-87.917,172.727,32.314,155.982
C06065=1060.855,212.254,-87.943,172.729,32.319,155.982
C06066=1060.861,212.503,-87.968,172.732,32.323,155.983
C06067=1060.867,212.752,-87.994,172.734,32.327,155.984
C06068=1060.873,213.000,-88.020,172.736,32.331,155.985
C06069=1060.879,213.248,-88.046,172.738,32.335,155.985
C06070=1060.885,213.497,-88.072,172.740,32.339,155.986
C06071=1060.891,213.745,-88.098,172.741,32.343,155.987
C06072=1060.897,213.994,-88.124,172.743,32.347,155.988
C06073=1060.903,214.242,-88.150,172.745,32.351,155.988
C06074=1060.909,214.491,-88.175,172.747,32.355,155.989
C06075=1060.916,214.740,-88.202,172.749,32.359,155.990
C06076=1060.921,214.989,-88.228,172.751,32.363,155.991
C06077=1060.928,215.237,-88.254,172.753,32.367,155.991
C06078=1060.934,215.485,-88.281,172.755,32.371,155.992
C06079=1060.940,215.734,-88.306,172.758,32.375,155.993
C06080=1060.946,215.983,-88.333,172.760,32.379,155.993
C06081=1060.952,216.231,-88.358,172.762,32.383,155.994
C06082=1060.957,216.480,-88.385,172.764,32.387,155.995
C06083=1060.964,216.729,-88.410,172.766,32.391,155.996
C06084=1060.970,216.977,-88.437,172.767,32.395,155.996
C06085=1060.976,217.226,-88.462,172.769,32.399,155.997
C06086=1060.982,217.474,-88.489,172.771,32.403,155.998
C06087=1060.989,217.722,-88.515,172.773,32.407,155.999
C06088=1060.994,217.971,-88.541,172.775,32.411,155.999
C06089=1061.001,218.220,-88.567,172.778,32.415,156.000
C06090=1061.007,218.468,-88.594,172.780,32.419,156.001
C06091=1061.013,218.717,-88.619,172.782,32.423,156.002
C06092=1061.019,218.965,-88.646,172.784,32.426,156.002
C06093=1061.025,219.214,-88.672,172.786,32.431,156.003
C06094=1061.031,219.463,-88.698,172.788,32.434,156.004
C06095=1061.038,219.711,-88.724,172.790,32.438,156.004
C06096=1061.044,219.960,-88.751,172.792,32.442,156.005
C06097=1061.050,220.208,-88.776,172.795,32.446,156.006
C06098=1061.056,220.457,-88.803,172.796,32.450,156.007
C06099=1061.062,220.706,-88.830,172.798,32.454,156.007
C06100=1061.069,220.954,-88.856,172.800,32.458,156.008
C06101=1061.075,221.185,-88.880,172.802,32.462,156.009
C06102=1061.080,221.417,-88.905,172.804,32.466,156.009
C06103=1061.085,221.648,-88.930,172.806,32.469,156.010
C06104=1061.091,221.880,-88.954,172.808,32.473,156.011
C06105=1061.097,222.112,-88.979,172.810,32.477,156.011
C06106=1061.103,222.343,-89.003,172.812,32.480,156.012
C06107=1061.108,222.574,-89.029,172.814,32.484,156.013
C06108=1061.113,222.805,-89.053,172.816,32.488,156.014
C06109=1061.120,223.053,-89.079,172.818,32.491,156.014
C06110=1061.126,223.303,-89.106,172.820,32.496,156.015
C06111=1061.132,223.551,-89.132,172.822,32.499,156.016
C06112=1061.137,223.800,-89.159,172.824,32.503,156.016
C06113=1061.144,224.048,-89.185,172.827,32.507,156.017
C06114=1061.150,224.297,-89.212,172.829,32.512,156.018
C06115=1061.156,224.545,-89.239,172.830,32.515,156.019
C06116=1061.162,224.794,-89.265,172.832,32.519,156.019
C06117=1061.168,225.042,-89.292,172.834,32.523,156.020
C06118=1061.175,225.291,-89.318,172.836,32.527,156.021
C06119=1061.181,225.539,-89.345,172.839,32.531,156.022
C06120=1061.186,225.788,-89.372,172.841,32.535,156.022
C06121=1061.193,226.037,-89.399,172.843,32.539,156.023
C06122=1061.198,226.285,-89.425,172.845,32.543,156.024
C06123=1061.205,226.533,-89.451,172.847,32.546,156.024
C06124=1061.211,226.782,-89.478,172.850,32.551,156.025
C06125=1061.217,227.030,-89.505,172.852,32.554,156.026
C06126=1061.223,227.279,-89.532,172.854,32.558,156.027
C06127=1061.230,227.527,-89.559,172.856,32.562,156.027
C06128=1061.235,227.776,-89.586,172.858,32.566,156.028
C06129=1061.242,228.024,-89.612,172.861,32.570,156.029
C06130=1061.248,228.273,-89.639,172.863,32.574,156.030
C06131=1061.254,228.521,-89.666,172.865,32.578,156.030
C06132=1061.260,228.770,-89.693,172.867,32.581,156.031
C06133=1061.266,229.018,-89.719,172.869,32.586,156.032
C06134=1061.273,229.268,-89.746,172.871,32.589,156.032
C06135=1061.279,229.515,-89.773,172.873,32.593,156.033
C06136=1061.285,229.763,-89.800,172.875,32.597,156.034
C06137=1061.291,230.013,-89.827,172.877,32.601,156.035
C06138=1061.297,230.261,-89.854,172.879,32.605,156.035
C06139=1061.303,230.509,-89.882,172.882,32.609,156.036
C06140=1061.309,230.758,-89.909,172.884,32.613,156.037
C06141=1061.315,231.006,-89.935,172.886,32.617,156.038
C06142=1061.321,231.255,-89.962,172.888,32.621,156.038
C06143=1061.327,231.503,-89.990,172.891,32.625,156.039
C06144=1061.334,231.752,-90.017,172.893,32.629,156.040
C06145=1061.339,232.000,-90.043,172.895,32.633,156.040
C06146=1061.345,232.248,-90.071,172.897,32.637,156.041
C06147=1061.352,232.497,-90.098,172.900,32.640,156.042
C06148=1061.358,232.746,-90.124,172.902,32.645,156.043
C06149=1061.364,232.994,-90.152,172.904,32.648,156.043
C06150=1061.370,233.242,-90.179,172.906,32.652,156.044
C06151=1061.376,233.491,-90.206,172.908,32.656,156.045
C06152=1061.382,233.739,-90.234,172.911,32.660,156.045
C06153=1061.388,233.989,-90.261,172.913,32.664,156.046
C06154=1061.394,234.236,-90.288,172.915,32.668,156.047
C06155=1061.401,234.485,-90.315,172.917,32.672,156.048
C06156=1061.407,234.733,-90.342,172.920,32.676,156.048
C06157=1061.412,234.960,-90.368,172.921,32.680,156.049
C06158=1061.418,235.189,-90.392,172.923,32.683,156.050
C06159=1061.423,235.416,-90.417,172.925,32.686,156.050
C06160=1061.429,235.644,-90.443,172.927,32.690,156.051
C06161=1061.434,235.871,-90.467,172.929,32.694,156.052
C06162=1061.439,236.098,-90.492,172.931,32.697,156.052
C06163=1061.446,236.326,-90.517,172.933,32.701,156.053
C06164=1061.451,236.553,-90.543,172.935,32.705,156.054
C06165=1061.457,236.802,-90.570,172.938,32.708,156.054
C06166=1061.463,237.050,-90.597,172.940,32.712,156.055
C06167=1061.469,237.299,-90.625,172.942,32.716,156.056
C06168=1061.475,237.547,-90.652,172.944,32.720,156.057
C06169=1061.482,237.795,-90.680,172.947,32.724,156.057
C06170=1061.487,238.043,-90.706,172.949,32.728,156.058
C06171=1061.494,238.292,-90.734,172.951,32.732,156.059
C06172=1061.500,238.541,-90.762,172.954,32.735,156.059
C06173=1061.506,238.789,-90.789,172.956,32.740,156.060
C06174=1061.513,239.037,-90.817,172.958,32.743,156.061
C06175=1061.519,239.285,-90.844,172.961,32.747,156.062
C06176=1061.524,239.535,-90.872,172.963,32.751,156.062
C06177=1061.530,239.782,-90.899,172.965,32.755,156.063
C06178=1061.537,240.031,-90.927,172.967,32.758,156.064
C06179=1061.543,240.280,-90.954,172.970,32.763,156.065
C06180=1061.549,240.528,-90.982,172.972,32.766,156.065
C06181=1061.555,240.776,-91.009,172.974,32.770,156.066
C06182=1061.561,241.025,-91.038,172.977,32.774,156.067
C06183=1061.567,241.273,-91.065,172.979,32.778,156.067
C06184=1061.574,241.522,-91.092,172.981,32.782,156.068
C06185=1061.579,241.770,-91.120,172.984,32.786,156.069
C06186=1061.586,242.018,-91.148,172.986,32.790,156.070
C06187=1061.592,242.267,-91.176,172.988,32.793,156.070
C06188=1061.598,242.515,-91.204,172.991,32.797,156.071
C06189=1061.605,242.763,-91.231,172.993,32.801,156.072
C06190=1061.610,243.013,-91.259,172.995,32.805,156.073
C06191=1061.616,243.260,-91.286,172.998,32.809,156.073
C06192=1061.622,243.509,-91.315,173.000,32.813,156.074
C06193=1061.628,243.757,-91.342,173.002,32.817,156.075
C06194=1061.634,244.006,-91.370,173.004,32.821,156.075
C06195=1061.641,244.254,-91.398,173.006,32.825,156.076
C06196=1061.646,244.502,-91.426,173.008,32.829,156.077
C06197=1061.653,244.751,-91.454,173.011,32.833,156.078
C06198=1061.659,244.999,-91.482,173.013,32.836,156.078
C06199=1061.664,245.247,-91.510,173.015,32.840,156.079
C06200=1061.671,245.496,-91.538,173.018,32.844,156.080
C06201=1061.677,245.745,-91.566,173.020,32.848,156.081
C06202=1061.683,245.993,-91.594,173.022,32.852,156.081
C06203=1061.689,246.241,-91.622,173.025,32.856,156.082
C06204=1061.696,246.490,-91.649,173.027,32.859,156.083
C06205=1061.701,246.738,-91.678,173.030,32.864,156.083
C06206=1061.707,246.986,-91.706,173.032,32.867,156.084
C06207=1061.713,247.234,-91.735,173.034,32.872,156.085
C06208=1061.720,247.483,-91.763,173.037,32.875,156.086
C06209=1061.725,247.731,-91.790,173.039,32.880,156.086
C06210=1061.731,247.980,-91.819,173.041,32.883,156.087
C06211=1061.737,248.228,-91.847,173.044,32.888,156.088
C06212=1061.742,248.476,-91.875,173.046,32.891,156.089
C06213=1061.748,248.701,-91.901,173.048,32.895,156.089
C06214=1061.754,248.925,-91.927,173.050,32.898,156.090
C06215=1061.759,249.149,-91.952,173.053,32.902,156.091
C06216=1061.765,249.374,-91.978,173.055,32.905,156.091
C06217=1061.770,249.598,-92.003,173.057,32.909,156.092
C06218=1061.775,249.823,-92.028,173.059,32.913,156.093
C06219=1061.781,250.046,-92.054,173.061,32.916,156.093
C06220=1061.786,250.271,-92.080,173.063,32.919,156.094
C06221=1061.792,250.520,-92.108,173.066,32.924,156.095
C06222=1061.798,250.768,-92.136,173.068,32.927,156.095
C06223=1061.805,251.016,-92.165,173.071,32.932,156.096
C06224=1061.811,251.265,-92.193,173.073,32.935,156.097
C06225=1061.817,251.513,-92.221,173.075,32.939,156.098
C06226=1061.822,251.761,-92.250,173.078,32.943,156.098
C06227=1061.828,252.010,-92.278,173.080,32.947,156.099
C06228=1061.835,252.257,-92.307,173.083,32.950,156.100
C06229=1061.841,252.506,-92.335,173.085,32.955,156.101
C06230=1061.847,252.755,-92.363,173.087,32.958,156.101
C06231=1061.853,253.002,-92.392,173.090,32.963,156.102
C06232=1061.859,253.251,-92.420,173.092,32.966,156.103
C06233=1061.865,253.499,-92.450,173.095,32.970,156.103
C06234=1061.872,253.748,-92.477,173.097,32.974,156.104
C06235=1061.878,253.996,-92.506,173.100,32.978,156.105
C06236=1061.884,254.245,-92.535,173.102,32.982,156.106
C06237=1061.890,254.493,-92.564,173.105,32.986,156.106
C06238=1061.895,254.741,-92.592,173.107,32.989,156.107
C06239=1061.902,254.989,-92.621,173.109,32.993,156.108
C06240=1061.908,255.238,-92.649,173.112,32.997,156.109
C06241=1061.915,255.485,-92.677,173.114,33.001,156.109
C06242=1061.920,255.734,-92.706,173.117,33.005,156.110
C06243=1061.927,255.982,-92.735,173.119,33.009,156.111
C06244=1061.933,256.231,-92.763,173.122,33.013,156.111
C06245=1061.939,256.479,-92.792,173.124,33.016,156.112
C06246=1061.945,256.727,-92.821,173.127,33.021,156.113
C06247=1061.951,256.976,-92.850,173.129,33.024,156.114
C06248=1061.957,257.223,-92.878,173.132,33.028,156.114
C06249=1061.964,257.471,-92.907,173.134,33.032,156.115
C06250=1061.970,257.720,-92.935,173.137,33.036,156.116
C06251=1061.976,257.968,-92.964,173.139,33.040,156.117
C06252=1061.982,258.216,-92.993,173.142,33.043,156.117
C06253=1061.988,258.465,-93.021,173.144,33.047,156.118
C06254=1061.994,258.713,-93.050,173.147,33.051,156.119
C06255=1062.001,258.961,-93.079,173.149,33.055,156.119
C06256=1062.007,259.209,-93.109,173.152,33.059,156.120
C06257=1062.013,259.458,-93.137,173.154,33.063,156.121
C06258=1062.019,259.706,-93.166,173.157,33.066,156.122
C06259=1062.025,259.954,-93.195,173.159,33.070,156.122
C06260=1062.032,260.202,-93.223,173.162,33.074,156.123
C06261=1062.038,260.451,-93.252,173.164,33.078,156.124
C06262=1062.044,260.699,-93.281,173.167,33.082,156.124
C06263=1062.051,260.947,-93.310,173.169,33.086,156.125
C06264=1062.058,261.196,-93.339,173.172,33.090,156.126
C06265=1062.064,261.444,-93.368,173.175,33.093,156.127
C06266=1062.070,261.692,-93.397,173.178,33.097,156.127
C06267=1062.076,261.941,-93.426,173.180,33.101,156.128
C06268=1062.082,262.189,-93.455,173.183,33.105,156.129
C06269=1062.088,262.412,-93.481,173.185,33.108,156.129
C06270=1062.094,262.636,-93.507,173.187,33.111,156.130
C06271=1062.099,262.860,-93.533,173.190,33.115,156.131
C06272=1062.106,263.082,-93.560,173.192,33.118,156.131
C06273=1062.111,263.305,-93.585,173.194,33.122,156.132
C06274=1062.116,263.529,-93.611,173.197,33.126,156.133
C06275=1062.122,263.752,-93.638,173.199,33.129,156.133
C06276=1062.127,263.975,-93.664,173.201,33.132,156.134
C06277=1062.133,264.224,-93.694,173.204,33.136,156.135
C06278=1062.139,264.472,-93.723,173.206,33.140,156.136
C06279=1062.145,264.720,-93.752,173.209,33.144,156.136
C06280=1062.152,264.968,-93.781,173.211,33.148,156.137
C06281=1062.157,265.217,-93.810,173.214,33.152,156.138
C06282=1062.164,265.464,-93.840,173.216,33.156,156.139
C06283=1062.170,265.712,-93.869,173.219,33.160,156.139
C06284=1062.176,265.961,-93.899,173.221,33.163,156.140
C06285=1062.182,266.209,-93.928,173.224,33.167,156.141
C06286=1062.189,266.458,-93.957,173.227,33.171,156.141
C06287=1062.194,266.706,-93.987,173.229,33.175,156.142
C06288=1062.200,266.954,-94.016,173.232,33.179,156.143
C06289=1062.207,267.202,-94.046,173.234,33.183,156.144
C06290=1062.213,267.450,-94.075,173.237,33.187,156.144
C06291=1062.219,267.698,-94.104,173.239,33.191,156.145
C06292=1062.226,267.947,-94.134,173.242,33.195,156.146
C06293=1062.232,268.195,-94.163,173.245,33.199,156.147
C06294=1062.238,268.443,-94.193,173.247,33.202,156.147
C06295=1062.244,268.691,-94.222,173.250,33.206,156.148
C06296=1062.250,268.939,-94.252,173.252,33.210,156.149
C06297=1062.256,269.187,-94.282,173.255,33.214,156.150
C06298=1062.262,269.435,-94.311,173.258,33.218,156.150
C06299=1062.269,269.684,-94.341,173.260,33.222,156.151
C06300=1062.275,269.932,-94.370,173.263,33.226,156.152
C06301=1062.280,270.180,-94.400,173.265,33.229,156.153
C06302=1062.287,270.428,-94.430,173.269,33.234,156.153
C06303=1062.292,270.676,-94.459,173.272,33.237,156.154
C06304=1062.300,270.925,-94.489,173.274,33.242,156.155
C06305=1062.306,271.173,-94.519,173.277,33.245,156.156
C06306=1062.311,271.421,-94.548,173.279,33.249,156.156
C06307=1062.318,271.669,-94.578,173.282,33.253,156.157
C06308=1062.323,271.917,-94.608,173.285,33.257,156.158
C06309=1062.331,272.165,-94.638,173.287,33.261,156.159
C06310=1062.336,272.414,-94.667,173.290,33.265,156.159
C06311=1062.343,272.661,-94.697,173.293,33.269,156.160
C06312=1062.348,272.910,-94.727,173.295,33.273,156.161
C06313=1062.355,273.158,-94.757,173.298,33.277,156.162
C06314=1062.361,273.406,-94.787,173.300,33.280,156.162
C06315=1062.367,273.654,-94.817,173.303,33.285,156.163
C06316=1062.373,273.902,-94.847,173.306,33.288,156.164
C06317=1062.379,274.151,-94.877,173.308,33.292,156.165
C06318=1062.385,274.399,-94.907,173.311,33.296,156.165
C06319=1062.392,274.646,-94.937,173.314,33.300,156.166
C06320=1062.397,274.895,-94.966,173.316,33.304,156.167
C06321=1062.404,275.143,-94.996,173.319,33.308,156.168
C06322=1062.410,275.391,-95.027,173.322,33.312,156.168
C06323=1062.416,275.639,-95.056,173.324,33.316,156.169
C06324=1062.423,275.887,-95.087,173.327,33.320,156.170
C06325=1062.428,276.112,-95.114,173.330,33.323,156.170
C06326=1062.433,276.338,-95.141,173.333,33.327,156.171
C06327=1062.439,276.562,-95.168,173.335,33.331,156.172
C06328=1062.445,276.788,-95.196,173.338,33.334,156.173
C06329=1062.450,277.013,-95.224,173.340,33.338,156.173
C06330=1062.455,277.238,-95.251,173.342,33.341,156.174
C06331=1062.461,277.463,-95.278,173.345,33.345,156.175
C06332=1062.467,277.689,-95.305,173.347,33.348,156.175
C06333=1062.473,277.936,-95.336,173.350,33.352,156.176
C06334=1062.479,278.184,-95.366,173.353,33.356,156.177
C06335=1062.486,278.432,-95.396,173.355,33.360,156.178
C06336=1062.492,278.680,-95.427,173.358,33.364,156.178
C06337=1062.498,278.929,-95.457,173.361,33.368,156.179
C06338=1062.504,279.177,-95.487,173.363,33.372,156.180
C06339=1062.511,279.425,-95.517,173.366,33.376,156.181
C06340=1062.517,279.673,-95.547,173.369,33.380,156.181
C06341=1062.523,279.921,-95.578,173.371,33.384,156.182
C06342=1062.529,280.170,-95.608,173.374,33.388,156.183
C06343=1062.535,280.417,-95.639,173.377,33.392,156.184
C06344=1062.541,280.665,-95.669,173.381,33.396,156.184
C06345=1062.548,280.913,-95.699,173.383,33.400,156.185
C06346=1062.554,281.161,-95.730,173.386,33.404,156.186
C06347=1062.560,281.409,-95.760,173.389,33.408,156.187
C06348=1062.566,281.658,-95.791,173.391,33.412,156.187
C06349=1062.572,281.905,-95.822,173.394,33.416,156.188
C06350=1062.579,282.153,-95.853,173.397,33.420,156.189
C06351=1062.584,282.401,-95.883,173.400,33.424,156.190
C06352=1062.590,282.649,-95.913,173.402,33.427,156.190
C06353=1062.597,282.897,-95.944,173.405,33.432,156.191
C06354=1062.602,283.145,-95.974,173.408,33.436,156.192
C06355=1062.609,283.394,-96.005,173.411,33.440,156.193
C06356=1062.615,283.641,-96.036,173.413,33.444,156.194
C06357=1062.621,283.890,-96.067,173.416,33.448,156.194
C06358=1062.627,284.137,-96.097,173.419,33.452,156.195
C06359=1062.634,284.386,-96.128,173.422,33.456,156.196
C06360=1062.639,284.634,-96.158,173.425,33.459,156.197
C06361=1062.646,284.882,-96.190,173.428,33.464,156.197
C06362=1062.652,285.129,-96.220,173.431,33.468,156.198
C06363=1062.658,285.378,-96.251,173.434,33.472,156.199
C06364=1062.665,285.625,-96.282,173.436,33.476,156.200
C06365=1062.671,285.874,-96.312,173.439,33.479,156.201
C06366=1062.677,286.122,-96.343,173.442,33.484,156.201
C06367=1062.683,286.369,-96.374,173.445,33.488,156.202
C06368=1062.689,286.617,-96.405,173.447,33.491,156.203
C06369=1062.696,286.866,-96.435,173.450,33.496,156.204
C06370=1062.702,287.113,-96.466,173.453,33.499,156.204
C06371=1062.708,287.361,-96.497,173.456,33.503,156.205
C06372=1062.715,287.610,-96.528,173.460,33.508,156.206
C06373=1062.721,287.857,-96.559,173.462,33.511,156.207
C06374=1062.727,288.106,-96.590,173.465,33.515,156.208
C06375=1062.733,288.353,-96.621,173.468,33.520,156.208
C06376=1062.740,288.601,-96.651,173.471,33.523,156.209
C06377=1062.746,288.850,-96.683,173.474,33.528,156.210
C06378=1062.752,289.097,-96.714,173.476,33.532,156.211
C06379=1062.758,289.345,-96.745,173.479,33.535,156.211
C06380=1062.764,289.593,-96.776,173.482,33.540,156.212
C06381=1062.770,289.824,-96.805,173.485,33.543,156.213
C06382=1062.776,290.055,-96.834,173.487,33.547,156.214
C06383=1062.782,290.285,-96.863,173.490,33.551,156.214
C06384=1062.788,290.515,-96.892,173.492,33.555,156.215
C06385=1062.793,290.746,-96.921,173.496,33.558,156.216
C06386=1062.799,290.976,-96.950,173.499,33.562,156.217
C06387=1062.805,291.206,-96.979,173.501,33.566,156.217
C06388=1062.810,291.437,-97.007,173.504,33.570,156.218
C06389=1062.817,291.685,-97.039,173.507,33.574,156.219
C06390=1062.823,291.933,-97.071,173.510,33.578,156.220
C06391=1062.829,292.180,-97.102,173.512,33.582,156.220
C06392=1062.835,292.429,-97.133,173.515,33.586,156.221
C06393=1062.841,292.677,-97.165,173.518,33.590,156.222
C06394=1062.848,292.924,-97.196,173.521,33.594,156.223
C06395=1062.854,293.172,-97.227,173.524,33.598,156.224
C06396=1062.860,293.421,-97.258,173.528,33.602,156.224
C06397=1062.866,293.668,-97.289,173.530,33.606,156.225
C06398=1062.873,293.916,-97.321,173.533,33.610,156.226
C06399=1062.879,294.164,-97.353,173.536,33.615,156.227
C06400=1062.885,294.412,-97.384,173.539,33.618,156.228
C06401=1062.892,294.659,-97.415,173.542,33.622,156.228
C06402=1062.897,294.908,-97.447,173.545,33.627,156.229
C06403=1062.904,295.156,-97.478,173.548,33.631,156.230
C06404=1062.910,295.403,-97.509,173.551,33.635,156.231
C06405=1062.916,295.652,-97.541,173.553,33.639,156.232
C06406=1062.923,295.900,-97.573,173.557,33.643,156.232
C06407=1062.929,296.148,-97.605,173.560,33.647,156.233
C06408=1062.935,296.395,-97.636,173.563,33.651,156.234
C06409=1062.941,296.643,-97.668,173.566,33.655,156.235
C06410=1062.948,296.891,-97.699,173.569,33.660,156.236
C06411=1062.954,297.139,-97.731,173.572,33.663,156.236
C06412=1062.960,297.386,-97.762,173.575,33.667,156.237
C06413=1062.966,297.635,-97.794,173.578,33.672,156.238
C06414=1062.972,297.883,-97.826,173.580,33.676,156.239
C06415=1062.978,298.131,-97.859,173.583,33.680,156.240
C06416=1062.984,298.378,-97.890,173.587,33.685,156.241
C06417=1062.990,298.626,-97.922,173.590,33.689,156.241
C06418=1062.996,298.874,-97.954,173.593,33.693,156.242
C06419=1063.003,299.122,-97.986,173.596,33.697,156.243
C06420=1063.008,299.370,-98.017,173.599,33.702,156.244
C06421=1063.015,299.617,-98.050,173.602,33.706,156.245
C06422=1063.021,299.865,-98.082,173.605,33.710,156.246
C06423=1063.027,300.113,-98.114,173.608,33.714,156.246
C06424=1063.033,300.361,-98.145,173.611,33.718,156.247
C06425=1063.039,300.608,-98.178,173.614,33.722,156.248
C06426=1063.045,300.857,-98.210,173.617,33.727,156.249
C06427=1063.052,301.104,-98.241,173.620,33.731,156.250
C06428=1063.058,301.352,-98.274,173.623,33.735,156.251
C06429=1063.063,301.600,-98.306,173.626,33.739,156.251
C06430=1063.069,301.848,-98.338,173.629,33.743,156.252
C06431=1063.076,302.095,-98.371,173.632,33.748,156.253
C06432=1063.082,302.343,-98.402,173.635,33.752,156.254
C06433=1063.089,302.591,-98.435,173.639,33.756,156.255
C06434=1063.095,302.839,-98.467,173.642,33.760,156.256
C06435=1063.101,303.087,-98.499,173.645,33.764,156.256
C06436=1063.108,303.335,-98.531,173.648,33.768,156.257
C06437=1063.113,303.573,-98.562,173.651,33.773,156.258
C06438=1063.119,303.811,-98.593,173.653,33.777,156.259
C06439=1063.125,304.049,-98.624,173.656,33.781,156.260
C06440=1063.131,304.287,-98.655,173.659,33.784,156.260
C06441=1063.137,304.524,-98.686,173.663,33.789,156.261
C06442=1063.143,304.763,-98.717,173.666,33.793,156.262
C06443=1063.148,305.001,-98.748,173.669,33.797,156.263
C06444=1063.155,305.239,-98.779,173.672,33.801,156.264
C06445=1063.161,305.487,-98.811,173.675,33.805,156.265
C06446=1063.168,305.735,-98.843,173.678,33.810,156.265
C06447=1063.174,305.982,-98.876,173.681,33.814,156.266
C06448=1063.180,306.231,-98.908,173.684,33.818,156.267
C06449=1063.187,306.478,-98.941,173.688,33.822,156.268
C06450=1063.193,306.726,-98.974,173.691,33.826,156.269
C06451=1063.199,306.974,-99.006,173.694,33.830,156.270
C06452=1063.206,307.221,-99.038,173.697,33.835,156.270
C06453=1063.212,307.469,-99.071,173.700,33.839,156.271
C06454=1063.218,307.717,-99.103,173.703,33.843,156.272
C06455=1063.225,307.965,-99.135,173.706,33.848,156.273
C06456=1063.231,308.212,-99.168,173.710,33.852,156.274
C06457=1063.237,308.460,-99.201,173.713,33.856,156.275
C06458=1063.243,308.708,-99.233,173.716,33.860,156.275
C06459=1063.249,308.956,-99.266,173.719,33.864,156.276
C06460=1063.256,309.203,-99.298,173.722,33.869,156.277
C06461=1063.263,309.450,-99.330,173.725,33.873,156.278
C06462=1063.270,309.699,-99.364,173.728,33.877,156.279
C06463=1063.276,309.946,-99.396,173.732,33.882,156.280
C06464=1063.282,310.195,-99.428,173.735,33.886,156.281
C06465=1063.288,310.442,-99.461,173.738,33.890,156.281
C06466=1063.294,310.690,-99.494,173.741,33.894,156.282
C06467=1063.301,310.937,-99.527,173.744,33.899,156.283
C06468=1063.308,311.186,-99.560,173.748,33.903,156.284
C06469=1063.314,311.433,-99.592,173.751,33.907,156.285
C06470=1063.321,311.681,-99.625,173.755,33.911,156.286
C06471=1063.327,311.928,-99.657,173.758,33.915,156.287
C06472=1063.334,312.176,-99.690,173.761,33.920,156.287
C06473=1063.340,312.424,-99.723,173.764,33.924,156.288
C06474=1063.347,312.672,-99.756,173.767,33.928,156.289
C06475=1063.353,312.919,-99.789,173.770,33.933,156.290
C06476=1063.359,313.167,-99.821,173.773,33.937,156.291
C06477=1063.366,313.415,-99.854,173.777,33.941,156.292
C06478=1063.373,313.663,-99.887,173.780,33.946,156.293
C06479=1063.379,313.910,-99.920,173.784,33.950,156.293
C06480=1063.385,314.158,-99.953,173.787,33.954,156.294
C06481=1063.392,314.406,-99.987,173.790,33.959,156.295
C06482=1063.398,314.653,-100.020,173.793,33.963,156.296
C06483=1063.403,314.901,-100.053,173.797,33.968,156.297
C06484=1063.410,315.149,-100.086,173.800,33.972,156.298
C06485=1063.416,315.396,-100.120,173.803,33.976,156.299
C06486=1063.422,315.644,-100.153,173.806,33.981,156.300
C06487=1063.429,315.892,-100.186,173.809,33.985,156.301
C06488=1063.434,316.140,-100.219,173.812,33.990,156.302
C06489=1063.441,316.387,-100.253,173.816,33.994,156.302
C06490=1063.446,316.635,-100.286,173.820,33.999,156.303
C06491=1063.453,316.883,-100.319,173.823,34.003,156.304
C06492=1063.459,317.130,-100.353,173.826,34.008,156.305
C06493=1063.465,317.370,-100.385,173.829,34.012,156.306
C06494=1063.471,317.610,-100.418,173.833,34.017,156.307
C06495=1063.478,317.850,-100.450,173.836,34.021,156.308
C06496=1063.484,318.090,-100.483,173.839,34.025,156.309
C06497=1063.490,318.330,-100.514,173.842,34.030,156.310
C06498=1063.495,318.569,-100.547,173.845,34.034,156.310
C06499=1063.501,318.810,-100.580,173.848,34.038,156.311
C06500=1063.508,319.050,-100.612,173.852,34.043,156.312
C06501=1063.513,319.297,-100.645,173.855,34.047,156.313
C06502=1063.521,319.545,-100.679,173.858,34.051,156.314
C06503=1063.526,319.793,-100.713,173.862,34.056,156.315
C06504=1063.533,320.040,-100.746,173.865,34.060,156.316
C06505=1063.539,320.288,-100.780,173.868,34.065,156.317
C06506=1063.546,320.536,-100.813,173.872,34.070,156.318
C06507=1063.552,320.784,-100.848,173.875,34.074,156.319
C06508=1063.558,321.031,-100.880,173.878,34.078,156.320
C06509=1063.564,321.278,-100.914,173.882,34.083,156.320
C06510=1063.571,321.526,-100.948,173.885,34.087,156.321
C06511=1063.577,321.774,-100.982,173.889,34.092,156.322
C06512=1063.584,322.022,-101.015,173.892,34.097,156.323
C06513=1063.590,322.269,-101.049,173.895,34.101,156.324
C06514=1063.597,322.517,-101.083,173.899,34.106,156.325
C06515=1063.603,322.765,-101.117,173.902,34.110,156.326
C06516=1063.609,323.013,-101.151,173.906,34.115,156.327
C06517=1063.616,323.260,-101.185,173.909,34.119,156.328
C06518=1063.622,323.508,-101.219,173.912,34.124,156.329
C06519=1063.629,323.755,-101.252,173.916,34.129,156.330
C06520=1063.635,324.003,-101.286,173.919,34.133,156.331
C06521=1063.642,324.250,-101.320,173.923,34.137,156.332
C06522=1063.648,324.498,-101.354,173.926,34.142,156.332
C06523=1063.654,324.745,-101.388,173.929,34.147,156.333
C06524=1063.661,324.993,-101.422,173.933,34.151,156.334
C06525=1063.667,325.240,-101.456,173.936,34.156,156.335
C06526=1063.674,325.489,-101.489,173.940,34.160,156.336
C06527=1063.680,325.736,-101.523,173.943,34.165,156.337
C06528=1063.686,325.984,-101.557,173.947,34.170,156.338
C06529=1063.693,326.232,-101.591,173.950,34.174,156.339
C06530=1063.699,326.479,-101.625,173.953,34.178,156.340
C06531=1063.706,326.726,-101.659,173.958,34.183,156.341
C06532=1063.713,326.974,-101.694,173.961,34.188,156.342
C06533=1063.719,327.222,-101.728,173.964,34.193,156.343
C06534=1063.726,327.469,-101.761,173.967,34.197,156.344
C06535=1063.733,327.717,-101.797,173.972,34.201,156.345
C06536=1063.739,327.964,-101.830,173.975,34.206,156.346
C06537=1063.746,328.212,-101.864,173.978,34.211,156.347
C06538=1063.752,328.460,-101.899,173.981,34.215,156.348
C06539=1063.759,328.707,-101.932,173.985,34.220,156.349
C06540=1063.765,328.955,-101.967,173.989,34.225,156.349
C06541=1063.772,329.203,-102.001,173.992,34.229,156.350
C06542=1063.779,329.449,-102.035,173.996,34.234,156.351
C06543=1063.785,329.697,-102.070,173.999,34.239,156.352
C06544=1063.792,329.945,-102.104,174.003,34.243,156.353
C06545=1063.799,330.193,-102.138,174.007,34.248,156.354
C06546=1063.805,330.441,-102.172,174.010,34.252,156.355
C06547=1063.811,330.687,-102.207,174.013,34.257,156.356
C06548=1063.818,330.935,-102.242,174.017,34.262,156.357
C06549=1063.824,331.173,-102.275,174.021,34.266,156.358
C06550=1063.830,331.409,-102.308,174.024,34.271,156.359
C06551=1063.836,331.647,-102.341,174.027,34.276,156.360
C06552=1063.842,331.884,-102.374,174.030,34.280,156.361
C06553=1063.849,332.121,-102.407,174.035,34.285,156.362
C06554=1063.855,332.357,-102.440,174.038,34.289,156.363
C06555=1063.861,332.595,-102.474,174.041,34.294,156.364
C06556=1063.867,332.831,-102.507,174.044,34.298,156.365
C06557=1063.874,333.079,-102.542,174.048,34.303,156.366
C06558=1063.880,333.327,-102.576,174.052,34.308,156.367
C06559=1063.887,333.574,-102.611,174.055,34.313,156.368
C06560=1063.893,333.821,-102.645,174.059,34.318,156.369
C06561=1063.900,334.069,-102.681,174.063,34.322,156.370
C06562=1063.906,334.317,-102.715,174.066,34.328,156.371
C06563=1063.913,334.564,-102.750,174.070,34.332,156.372
C06564=1063.920,334.811,-102.785,174.073,34.337,156.373
C06565=1063.926,335.059,-102.820,174.077,34.342,156.374
C06566=1063.932,335.306,-102.854,174.081,34.347,156.375
C06567=1063.939,335.553,-102.890,174.084,34.351,156.376
C06568=1063.945,335.802,-102.925,174.088,34.356,156.377
C06569=1063.951,336.049,-102.960,174.092,34.361,156.378
C06570=1063.958,336.296,-102.995,174.095,34.366,156.379
C06571=1063.965,336.544,-103.029,174.099,34.371,156.380
C06572=1063.971,336.792,-103.064,174.102,34.376,156.381
C06573=1063.978,337.039,-103.100,174.107,34.381,156.382
C06574=1063.985,337.286,-103.135,174.110,34.386,156.383
C06575=1063.991,337.533,-103.169,174.113,34.390,156.384
C06576=1063.997,337.781,-103.205,174.117,34.396,156.385
C06577=1064.004,338.029,-103.240,174.121,34.400,156.386
C06578=1064.010,338.276,-103.275,174.125,34.406,156.387
C06579=1064.016,338.524,-103.310,174.128,34.410,156.388
C06580=1064.023,338.771,-103.346,174.132,34.415,156.389
C06581=1064.030,339.019,-103.381,174.136,34.421,156.390
C06582=1064.036,339.266,-103.416,174.139,34.425,156.391
C06583=1064.043,339.514,-103.452,174.143,34.430,156.392
C06584=1064.050,339.761,-103.487,174.147,34.435,156.393
C06585=1064.056,340.008,-103.522,174.151,34.440,156.394
C06586=1064.062,340.256,-103.558,174.154,34.445,156.396
C06587=1064.069,340.503,-103.593,174.159,34.450,156.397
C06588=1064.076,340.751,-103.628,174.162,34.455,156.398
C06589=1064.082,340.998,-103.664,174.166,34.461,156.399
C06590=1064.089,341.245,-103.699,174.169,34.465,156.400
C06591=1064.096,341.492,-103.735,174.173,34.470,156.401
C06592=1064.102,341.740,-103.770,174.177,34.476,156.402
C06593=1064.109,341.988,-103.805,174.180,34.480,156.403
C06594=1064.115,342.235,-103.841,174.185,34.485,156.404
C06595=1064.122,342.482,-103.877,174.188,34.491,156.405
C06596=1064.128,342.729,-103.912,174.192,34.495,156.406
C06597=1064.134,342.977,-103.948,174.195,34.500,156.407
C06598=1064.141,343.224,-103.983,174.200,34.506,156.408
C06599=1064.148,343.471,-104.019,174.203,34.511,156.409
C06600=1064.155,343.719,-104.055,174.207,34.516,156.410
C06601=1064.162,343.967,-104.090,174.211,34.521,156.411
C06602=1064.168,344.214,-104.127,174.215,34.526,156.413
C06603=1064.175,344.461,-104.162,174.218,34.531,156.414
C06604=1064.181,344.709,-104.197,174.223,34.536,156.415
C06605=1064.187,344.944,-104.231,174.226,34.541,156.416
C06606=1064.193,345.178,-104.265,174.230,34.546,156.417
C06607=1064.200,345.413,-104.299,174.234,34.551,156.418
C06608=1064.206,345.648,-104.334,174.237,34.556,156.419
C06609=1064.212,345.882,-104.368,174.241,34.561,156.420
C06610=1064.219,346.116,-104.402,174.244,34.566,156.421
C06611=1064.225,346.351,-104.436,174.248,34.571,156.422
C06612=1064.231,346.586,-104.470,174.252,34.576,156.423
C06613=1064.237,346.834,-104.506,174.255,34.581,156.424
C06614=1064.244,347.080,-104.542,174.260,34.586,156.425
C06615=1064.250,347.327,-104.578,174.263,34.592,156.427
C06616=1064.258,347.575,-104.614,174.267,34.597,156.428
C06617=1064.264,347.822,-104.650,174.272,34.602,156.429
C06618=1064.270,348.069,-104.687,174.275,34.607,156.430
C06619=1064.276,348.317,-104.723,174.279,34.612,156.431
C06620=1064.284,348.565,-104.759,174.283,34.618,156.432
C06621=1064.290,348.812,-104.795,174.287,34.623,156.433
C06622=1064.297,349.059,-104.832,174.291,34.628,156.434
C06623=1064.304,349.306,-104.867,174.295,34.634,156.436
C06624=1064.311,349.554,-104.904,174.299,34.639,156.437
C06625=1064.317,349.801,-104.940,174.302,34.644,156.438
C06626=1064.323,350.048,-104.976,174.307,34.650,156.439
C06627=1064.330,350.295,-105.012,174.311,34.655,156.440
C06628=1064.337,350.542,-105.049,174.315,34.661,156.441
C06629=1064.343,350.790,-105.085,174.319,34.666,156.442
C06630=1064.350,351.037,-105.121,174.322,34.671,156.444
C06631=1064.357,351.285,-105.158,174.327,34.676,156.445
C06632=1064.364,351.532,-105.194,174.331,34.682,156.446
C06633=1064.371,351.779,-105.231,174.334,34.687,156.447
C06634=1064.377,352.026,-105.267,174.339,34.693,156.448
C06635=1064.383,352.274,-105.304,174.343,34.698,156.449
C06636=1064.391,352.521,-105.340,174.346,34.704,156.451
C06637=1064.397,352.768,-105.376,174.351,34.709,156.452
C06638=1064.404,353.014,-105.414,174.355,34.714,156.453
C06639=1064.411,353.262,-105.450,174.359,34.720,156.454
C06640=1064.417,353.509,-105.487,174.363,34.725,156.455
C06641=1064.423,353.756,-105.523,174.367,34.731,156.456
C06642=1064.430,354.004,-105.560,174.371,34.736,156.458
C06643=1064.437,354.251,-105.596,174.375,34.742,156.459
C06644=1064.444,354.498,-105.634,174.379,34.747,156.460
C06645=1064.450,354.745,-105.670,174.383,34.753,156.461
C06646=1064.457,354.993,-105.707,174.387,34.758,156.462
C06647=1064.464,355.240,-105.744,174.392,34.764,156.464
C06648=1064.470,355.487,-105.781,174.395,34.769,156.465
C06649=1064.477,355.734,-105.818,174.399,34.775,156.466
C06650=1064.484,355.981,-105.855,174.404,34.780,156.467
C06651=1064.491,356.229,-105.892,174.407,34.786,156.468
C06652=1064.497,356.476,-105.928,174.412,34.792,156.470
C06653=1064.504,356.723,-105.966,174.416,34.797,156.471
C06654=1064.511,356.970,-106.002,174.420,34.803,156.472
C06655=1064.518,357.217,-106.040,174.424,34.808,156.473
C06656=1064.525,357.465,-106.076,174.428,34.814,156.475
C06657=1064.531,357.711,-106.114,174.433,34.820,156.476
C06658=1064.538,357.959,-106.150,174.437,34.825,156.477
C06659=1064.545,358.205,-106.188,174.440,34.831,156.478
C06660=1064.552,358.453,-106.224,174.445,34.837,156.479
C06661=1064.558,358.689,-106.260,174.449,34.842,156.481
C06662=1064.565,358.927,-106.296,174.453,34.847,156.482
C06663=1064.571,359.163,-106.332,174.457,34.853,156.483
C06664=1064.578,359.400,-106.367,174.461,34.858,156.484
C06665=1064.584,359.636,-106.403,174.465,34.864,156.485
C06666=1064.591,359.873,-106.438,174.469,34.869,156.487
C06667=1064.597,360.110,-106.475,174.473,34.875,156.488
C06668=1064.603,360.346,-106.510,174.477,34.880,156.489
C06669=1064.610,360.594,-106.548,174.482,34.886,156.490
C06670=1064.618,360.841,-106.585,174.486,34.892,156.492
C06671=1064.624,361.087,-106.622,174.489,34.897,156.493
C06672=1064.631,361.335,-106.660,174.494,34.903,156.494
C06673=1064.638,361.582,-106.697,174.498,34.909,156.495
C06674=1064.644,361.829,-106.734,174.503,34.915,156.497
C06675=1064.652,362.076,-106.772,174.507,34.921,156.498
C06676=1064.658,362.323,-106.810,174.511,34.926,156.499
C06677=1064.665,362.570,-106.847,174.515,34.933,156.501
C06678=1064.672,362.817,-106.885,174.520,34.938,156.502
C06679=1064.678,363.064,-106.923,174.524,34.944,156.503
C06680=1064.686,363.312,-106.960,174.529,34.950,156.504
C06681=1064.692,363.558,-106.997,174.533,34.956,156.506
C06682=1064.699,363.805,-107.036,174.536,34.961,156.507
C06683=1064.706,364.053,-107.073,174.541,34.968,156.508
C06684=1064.713,364.300,-107.111,174.545,34.973,156.510
C06685=1064.719,364.546,-107.148,174.550,34.980,156.511
C06686=1064.727,364.793,-107.187,174.554,34.985,156.512
C06687=1064.733,365.040,-107.225,174.559,34.991,156.514
C06688=1064.741,365.288,-107.262,174.563,34.998,156.515
C06689=1064.746,365.534,-107.300,174.567,35.003,156.516
C06690=1064.754,365.781,-107.338,174.571,35.010,156.518
C06691=1064.760,366.028,-107.376,174.576,35.016,156.519
C06692=1064.767,366.276,-107.415,174.580,35.021,156.520
C06693=1064.774,366.523,-107.452,174.585,35.028,156.522
C06694=1064.780,366.769,-107.491,174.589,35.034,156.523
C06695=1064.788,367.016,-107.528,174.594,35.039,156.524
C06696=1064.794,367.263,-107.567,174.598,35.046,156.526
C06697=1064.802,367.510,-107.604,174.603,35.052,156.527
C06698=1064.808,367.757,-107.643,174.606,35.058,156.528
C06699=1064.815,368.004,-107.681,174.611,35.064,156.530
C06700=1064.822,368.251,-107.719,174.615,35.070,156.531
C06701=1064.829,368.498,-107.758,174.620,35.076,156.532
C06702=1064.836,368.745,-107.795,174.624,35.082,156.534
C06703=1064.843,368.991,-107.834,174.629,35.088,156.535
C06704=1064.849,369.238,-107.873,174.633,35.095,156.537
C06705=1064.857,369.485,-107.910,174.638,35.101,156.538
C06706=1064.863,369.732,-107.949,174.642,35.107,156.539
C06707=1064.871,369.979,-107.986,174.647,35.113,156.541
C06708=1064.877,370.226,-108.025,174.652,35.119,156.542
C06709=1064.884,370.473,-108.064,174.656,35.126,156.543
C06710=1064.892,370.720,-108.102,174.661,35.132,156.545
C06711=1064.898,370.967,-108.141,174.665,35.138,156.546
C06712=1064.905,371.214,-108.179,174.670,35.145,156.548
C06713=1064.913,371.460,-108.218,174.674,35.151,156.549
C06714=1064.920,371.707,-108.256,174.679,35.157,156.551
C06715=1064.927,371.954,-108.294,174.683,35.163,156.552
C06716=1064.934,372.202,-108.333,174.688,35.169,156.553
C06717=1064.944,372.551,-108.387,174.695,35.178,156.555
C06718=1064.954,372.899,-108.443,174.700,35.187,156.557
C06719=1064.964,373.248,-108.497,174.707,35.196,156.559
C06720=1064.973,373.596,-108.553,174.714,35.206,156.562
C06721=1064.980,373.843,-108.591,174.719,35.212,156.563
C06722=1064.987,374.089,-108.630,174.723,35.219,156.564
C06723=1064.994,374.336,-108.668,174.728,35.225,156.566
C06724=1065.001,374.583,-108.707,174.732,35.232,156.567
C06725=1065.008,374.831,-108.746,174.737,35.238,156.569
C06726=1065.015,375.077,-108.785,174.742,35.244,156.570
C06727=1065.022,375.324,-108.824,174.746,35.251,156.572
C06728=1065.029,375.570,-108.864,174.751,35.257,156.573
C06729=1065.036,375.817,-108.903,174.755,35.264,156.575
C06730=1065.043,376.064,-108.941,174.760,35.271,156.576
C06731=1065.050,376.311,-108.980,174.765,35.277,156.578
C06732=1065.057,376.558,-109.020,174.769,35.284,156.579
C06733=1065.068,376.947,-109.081,174.777,35.294,156.582
C06734=1065.079,377.336,-109.144,174.784,35.305,156.584
C06735=1065.090,377.725,-109.205,174.792,35.315,156.586
C06736=1065.102,378.113,-109.267,174.799,35.325,156.589
C06737=1065.109,378.361,-109.306,174.804,35.332,156.590
C06738=1065.116,378.607,-109.345,174.808,35.339,156.592
C06739=1065.123,378.854,-109.384,174.814,35.345,156.593
C06740=1065.131,379.101,-109.424,174.819,35.352,156.595
C06741=1065.138,379.347,-109.464,174.823,35.359,156.596
C06742=1065.145,379.594,-109.503,174.828,35.365,156.598
C06743=1065.152,379.841,-109.542,174.833,35.372,156.599
C06744=1065.158,380.088,-109.582,174.837,35.379,156.601
C06745=1065.166,380.334,-109.621,174.843,35.386,156.603
C06746=1065.173,380.581,-109.661,174.848,35.393,156.604
C06747=1065.180,380.828,-109.700,174.852,35.399,156.606
C06748=1065.188,381.075,-109.740,174.857,35.406,156.607
C06749=1065.195,381.321,-109.780,174.862,35.413,156.609
C06750=1065.202,381.567,-109.819,174.867,35.420,156.610
C06751=1065.209,381.814,-109.860,174.872,35.427,156.612
C06752=1065.216,382.060,-109.899,174.877,35.434,156.614
C06753=1065.224,382.307,-109.939,174.882,35.441,156.615
C06754=1065.230,382.554,-109.979,174.886,35.448,156.617
C06755=1065.237,382.801,-110.018,174.892,35.455,156.618
C06756=1065.245,383.048,-110.058,174.897,35.462,156.620
C06757=1065.251,383.294,-110.098,174.901,35.469,156.622
C06758=1065.259,383.541,-110.138,174.906,35.476,156.623
C06759=1065.266,383.787,-110.178,174.912,35.483,156.625
C06760=1065.273,384.034,-110.219,174.916,35.490,156.626
C06761=1065.280,384.280,-110.259,174.921,35.497,156.628
C06762=1065.287,384.527,-110.299,174.926,35.504,156.630
C06763=1065.294,384.773,-110.339,174.932,35.511,156.631
C06764=1065.302,385.020,-110.379,174.936,35.519,156.633
C06765=1065.309,385.267,-110.419,174.941,35.525,156.635
C06766=1065.317,385.513,-110.459,174.946,35.532,156.636
C06767=1065.323,385.760,-110.499,174.952,35.540,156.638
C06768=1065.331,386.006,-110.539,174.956,35.547,156.640
C06769=1065.339,386.281,-110.584,174.962,35.555,156.642
C06770=1065.347,386.555,-110.629,174.968,35.563,156.643
C06771=1065.355,386.830,-110.674,174.973,35.571,156.645
C06772=1065.363,387.105,-110.718,174.979,35.579,156.647
C06773=1065.371,387.351,-110.760,174.985,35.586,156.649
C06774=1065.378,387.598,-110.799,174.989,35.594,156.651
C06775=1065.385,387.844,-110.840,174.994,35.601,156.652
C06776=1065.393,388.091,-110.880,175.000,35.608,156.654
C06777=1065.400,388.337,-110.921,175.005,35.615,156.656
C06778=1065.407,388.584,-110.961,175.010,35.623,156.657
C06779=1065.415,388.830,-111.002,175.015,35.630,156.659
C06780=1065.422,389.077,-111.042,175.020,35.637,156.661
C06781=1065.430,389.323,-111.082,175.026,35.645,156.663
C06782=1065.437,389.570,-111.124,175.031,35.652,156.664
C06783=1065.445,389.816,-111.164,175.036,35.660,156.666
C06784=1065.452,390.063,-111.205,175.041,35.667,156.668
C06785=1065.460,390.309,-111.246,175.046,35.674,156.669
C06786=1065.467,390.555,-111.286,175.052,35.682,156.671
C06787=1065.474,390.802,-111.327,175.057,35.689,156.673
C06788=1065.482,391.049,-111.368,175.063,35.697,156.675
C06789=1065.489,391.295,-111.409,175.067,35.704,156.676
C06790=1065.496,391.542,-111.450,175.072,35.712,156.678
C06791=1065.504,391.787,-111.490,175.078,35.719,156.680
C06792=1065.511,392.034,-111.531,175.083,35.727,156.682
C06793=1065.518,392.281,-111.573,175.089,35.735,156.684
C06794=1065.526,392.527,-111.614,175.094,35.742,156.685
C06795=1065.534,392.774,-111.655,175.100,35.750,156.687
C06796=1065.541,393.020,-111.696,175.105,35.758,156.689
C06797=1065.548,393.267,-111.737,175.110,35.766,156.691
C06798=1065.556,393.513,-111.778,175.115,35.773,156.693
C06799=1065.564,393.760,-111.819,175.121,35.781,156.695
C06800=1065.571,394.006,-111.861,175.126,35.788,156.696
C06801=1065.578,394.251,-111.902,175.132,35.796,156.698
C06802=1065.585,394.498,-111.943,175.137,35.804,156.700
C06803=1065.592,394.745,-111.984,175.143,35.812,156.702
C06804=1065.600,394.991,-112.026,175.148,35.820,156.704
C06805=1065.607,395.237,-112.067,175.154,35.828,156.706
C06806=1065.615,395.484,-112.109,175.159,35.835,156.708
C06807=1065.622,395.730,-112.151,175.165,35.844,156.709
C06808=1065.630,395.977,-112.192,175.170,35.851,156.711
C06809=1065.638,396.223,-112.233,175.175,35.859,156.713
C06810=1065.646,396.469,-112.275,175.181,35.867,156.715
C06811=1065.653,396.716,-112.316,175.186,35.875,156.717
C06812=1065.661,396.962,-112.358,175.192,35.883,156.719
C06813=1065.668,397.209,-112.399,175.197,35.891,156.721
C06814=1065.675,397.454,-112.441,175.203,35.899,156.723
C06815=1065.683,397.701,-112.482,175.208,35.907,156.725
C06816=1065.691,397.948,-112.525,175.214,35.915,156.727
C06817=1065.699,398.194,-112.567,175.220,35.923,156.728
C06818=1065.705,398.441,-112.608,175.225,35.931,156.730
C06819=1065.713,398.687,-112.650,175.231,35.940,156.732
C06820=1065.720,398.933,-112.692,175.237,35.948,156.734
C06821=1065.728,399.179,-112.735,175.242,35.956,156.736
C06822=1065.736,399.426,-112.776,175.248,35.964,156.738
C06823=1065.743,399.672,-112.818,175.253,35.973,156.740
C06824=1065.751,399.918,-112.860,175.259,35.981,156.742
C06825=1065.760,400.209,-112.910,175.267,35.991,156.745
C06826=1065.769,400.500,-112.960,175.273,36.000,156.747
C06827=1065.778,400.792,-113.009,175.280,36.010,156.749
C06828=1065.786,401.082,-113.059,175.286,36.020,156.752
C06829=1065.795,401.329,-113.101,175.292,36.029,156.754
C06830=1065.802,401.575,-113.143,175.298,36.037,156.756
C06831=1065.810,401.821,-113.185,175.303,36.045,156.758
C06832=1065.817,402.068,-113.228,175.309,36.053,156.760
C06833=1065.825,402.314,-113.270,175.316,36.062,156.762
C06834=1065.833,402.560,-113.313,175.322,36.070,156.764
C06835=1065.841,402.806,-113.355,175.327,36.079,156.766
C06836=1065.848,403.053,-113.398,175.333,36.088,156.768
C06837=1065.856,403.299,-113.440,175.339,36.096,156.770
C06838=1065.864,403.545,-113.483,175.345,36.104,156.772
C06839=1065.871,403.791,-113.525,175.350,36.113,156.774
C06840=1065.879,404.038,-113.568,175.356,36.122,156.776
C06841=1065.887,404.283,-113.610,175.362,36.130,156.778
C06842=1065.895,404.530,-113.653,175.369,36.139,156.781
C06843=1065.903,404.775,-113.696,175.375,36.147,156.783
C06844=1065.910,405.022,-113.739,175.381,36.157,156.785
C06845=1065.918,405.268,-113.781,175.386,36.165,156.787
C06846=1065.926,405.515,-113.824,175.392,36.174,156.789
C06847=1065.933,405.760,-113.867,175.398,36.183,156.791
C06848=1065.941,406.007,-113.910,175.405,36.192,156.793
C06849=1065.949,406.253,-113.953,175.411,36.200,156.796
C06850=1065.956,406.499,-113.996,175.417,36.209,156.798
C06851=1065.965,406.745,-114.039,175.423,36.218,156.800
C06852=1065.972,406.991,-114.082,175.428,36.227,156.802
C06853=1065.980,407.237,-114.126,175.435,36.236,156.804
C06854=1065.988,407.483,-114.169,175.441,36.245,156.807
C06855=1065.995,407.730,-114.211,175.447,36.254,156.809
C06856=1066.003,407.976,-114.255,175.453,36.263,156.811
C06857=1066.011,408.222,-114.298,175.460,36.272,156.813
C06858=1066.019,408.469,-114.341,175.466,36.281,156.815
C06859=1066.026,408.714,-114.385,175.472,36.290,156.818
C06860=1066.035,408.960,-114.428,175.478,36.299,156.820
C06861=1066.043,409.207,-114.471,175.485,36.308,156.822
C06862=1066.050,409.453,-114.515,175.491,36.317,156.824
C06863=1066.058,409.698,-114.558,175.497,36.327,156.827
C06864=1066.066,409.945,-114.601,175.504,36.336,156.829
C06865=1066.074,410.191,-114.645,175.510,36.345,156.831
C06866=1066.082,410.437,-114.689,175.516,36.354,156.834
C06867=1066.090,410.683,-114.732,175.522,36.364,156.836
C06868=1066.098,410.929,-114.776,175.529,36.373,156.838
C06869=1066.106,411.176,-114.819,175.535,36.382,156.840
C06870=1066.115,411.421,-114.863,175.541,36.392,156.843
C06871=1066.122,411.667,-114.906,175.548,36.401,156.845
C06872=1066.130,411.913,-114.950,175.554,36.411,156.847
C06873=1066.138,412.159,-114.994,175.560,36.420,156.850
C06874=1066.146,412.405,-115.037,175.568,36.429,156.852
C06875=1066.154,412.651,-115.082,175.574,36.439,156.854
C06876=1066.162,412.897,-115.125,175.581,36.448,156.857
C06877=1066.170,413.143,-115.170,175.587,36.458,156.859
C06878=1066.178,413.390,-115.214,175.593,36.467,156.862
C06879=1066.187,413.635,-115.257,175.600,36.477,156.864
C06880=1066.195,413.882,-115.301,175.607,36.486,156.866
C06881=1066.204,414.176,-115.354,175.615,36.498,156.869
C06882=1066.215,414.472,-115.407,175.623,36.510,156.872
C06883=1066.224,414.767,-115.460,175.630,36.522,156.875
C06884=1066.234,415.063,-115.513,175.639,36.533,156.878
C06885=1066.241,415.309,-115.558,175.646,36.543,156.880
C06886=1066.249,415.555,-115.602,175.652,36.553,156.883
C06887=1066.258,415.801,-115.646,175.659,36.562,156.885
C06888=1066.266,416.046,-115.691,175.666,36.573,156.888
C06889=1066.274,416.293,-115.735,175.673,36.582,156.890
C06890=1066.282,416.539,-115.780,175.679,36.592,156.893
C06891=1066.290,416.784,-115.824,175.686,36.602,156.895
C06892=1066.299,417.030,-115.868,175.693,36.612,156.898
C06893=1066.307,417.276,-115.914,175.700,36.622,156.900
C06894=1066.316,417.522,-115.958,175.706,36.632,156.903
C06895=1066.323,417.768,-116.003,175.714,36.642,156.906
C06896=1066.331,418.013,-116.047,175.720,36.652,156.908
C06897=1066.340,418.260,-116.092,175.728,36.663,156.911
C06898=1066.348,418.505,-116.137,175.735,36.673,156.913
C06899=1066.356,418.751,-116.181,175.741,36.683,156.916
C06900=1066.365,418.997,-116.226,175.749,36.693,156.918
C06901=1066.373,419.242,-116.271,175.755,36.703,156.921
C06902=1066.381,419.489,-116.316,175.763,36.714,156.924
C06903=1066.389,419.734,-116.361,175.770,36.724,156.926
C06904=1066.398,419.980,-116.406,175.776,36.734,156.929
C06905=1066.406,420.226,-116.451,175.784,36.744,156.931
C06906=1066.415,420.472,-116.496,175.791,36.755,156.934
C06907=1066.423,420.718,-116.542,175.798,36.765,156.937
C06908=1066.432,420.964,-116.587,175.805,36.776,156.940
C06909=1066.440,421.209,-116.631,175.813,36.786,156.942
C06910=1066.447,421.455,-116.677,175.819,36.797,156.945
C06911=1066.456,421.701,-116.722,175.827,36.807,156.948
C06912=1066.464,421.946,-116.768,175.835,36.818,156.950
C06913=1066.473,422.192,-116.813,175.842,36.829,156.953
C06914=1066.482,422.438,-116.859,175.849,36.839,156.956
C06915=1066.490,422.683,-116.905,175.856,36.850,156.959
C06916=1066.499,422.929,-116.950,175.864,36.861,156.961
C06917=1066.506,423.174,-116.996,175.871,36.871,156.964
C06918=1066.515,423.420,-117.041,175.879,36.882,156.967
C06919=1066.524,423.666,-117.087,175.886,36.893,156.970
C06920=1066.532,423.911,-117.132,175.893,36.904,156.972
C06921=1066.540,424.158,-117.178,175.901,36.915,156.975
C06922=1066.549,424.403,-117.224,175.909,36.926,156.978
C06923=1066.557,424.648,-117.270,175.916,36.936,156.981
C06924=1066.566,424.894,-117.315,175.924,36.947,156.984
C06925=1066.574,425.140,-117.361,175.931,36.958,156.986
C06926=1066.584,425.385,-117.407,175.939,36.969,156.989
C06927=1066.591,425.631,-117.453,175.946,36.980,156.992
C06928=1066.600,425.876,-117.499,175.954,36.991,156.995
C06929=1066.609,426.122,-117.545,175.962,37.003,156.998
C06930=1066.618,426.367,-117.591,175.970,37.014,157.001
C06931=1066.626,426.613,-117.637,175.977,37.025,157.004
C06932=1066.636,426.859,-117.684,175.985,37.036,157.007
C06933=1066.644,427.105,-117.730,175.993,37.047,157.010
C06934=1066.652,427.350,-117.776,176.001,37.059,157.013
C06935=1066.661,427.595,-117.822,176.009,37.070,157.016
C06936=1066.670,427.840,-117.869,176.017,37.081,157.018
C06937=1066.680,428.156,-117.928,176.026,37.096,157.022
C06938=1066.692,428.471,-117.987,176.037,37.111,157.026
C06939=1066.703,428.786,-118.048,176.047,37.126,157.030
C06940=1066.714,429.101,-118.107,176.057,37.141,157.034
C06941=1066.722,429.346,-118.154,176.065,37.152,157.037
C06942=1066.732,429.592,-118.201,176.073,37.164,157.040
C06943=1066.741,429.837,-118.248,176.082,37.176,157.043
C06944=1066.750,430.083,-118.294,176.090,37.187,157.046
C06945=1066.758,430.328,-118.341,176.098,37.199,157.049
C06946=1066.767,430.574,-118.388,176.106,37.210,157.052
C06947=1066.776,430.818,-118.435,176.114,37.222,157.055
C06948=1066.785,431.064,-118.481,176.122,37.234,157.059
C06949=1066.793,431.309,-118.528,176.130,37.246,157.062
C06950=1066.803,431.555,-118.576,176.139,37.258,157.065
C06951=1066.811,431.800,-118.623,176.147,37.270,157.068
C06952=1066.820,432.045,-118.670,176.155,37.282,157.071
C06953=1066.829,432.291,-118.717,176.163,37.294,157.074
C06954=1066.838,432.536,-118.764,176.172,37.306,157.078
C06955=1066.847,432.781,-118.812,176.180,37.318,157.081
C06956=1066.856,433.027,-118.859,176.189,37.330,157.084
C06957=1066.864,433.272,-118.907,176.197,37.343,157.087
C06958=1066.873,433.517,-118.954,176.206,37.355,157.091
C06959=1066.882,433.762,-119.002,176.214,37.367,157.094
C06960=1066.891,434.008,-119.049,176.222,37.379,157.097
C06961=1066.899,434.253,-119.096,176.232,37.392,157.100
C06962=1066.909,434.498,-119.144,176.240,37.404,157.104
C06963=1066.918,434.743,-119.192,176.249,37.416,157.107
C06964=1066.927,434.989,-119.239,176.257,37.429,157.110
C06965=1066.936,435.234,-119.287,176.266,37.442,157.114
C06966=1066.946,435.479,-119.335,176.275,37.454,157.117
C06967=1066.955,435.724,-119.383,176.283,37.466,157.121
C06968=1066.963,435.970,-119.431,176.293,37.479,157.124
C06969=1066.972,436.214,-119.479,176.301,37.492,157.127
C06970=1066.982,436.460,-119.526,176.310,37.505,157.131
C06971=1066.991,436.704,-119.575,176.319,37.517,157.134
C06972=1067.000,436.950,-119.622,176.328,37.530,157.138
C06973=1067.010,437.195,-119.671,176.337,37.543,157.141
C06974=1067.019,437.440,-119.718,176.346,37.555,157.145
C06975=1067.028,437.685,-119.767,176.355,37.568,157.148
C06976=1067.037,437.931,-119.815,176.364,37.582,157.152
C06977=1067.046,438.175,-119.863,176.373,37.594,157.155
C06978=1067.056,438.421,-119.911,176.382,37.607,157.159
C06979=1067.065,438.666,-119.960,176.392,37.621,157.162
C06980=1067.075,438.911,-120.009,176.401,37.633,157.166
C06981=1067.084,439.155,-120.057,176.410,37.647,157.169
C06982=1067.093,439.400,-120.106,176.419,37.660,157.173
C06983=1067.102,439.646,-120.154,176.429,37.673,157.177
C06984=1067.111,439.891,-120.203,176.437,37.687,157.180
C06985=1067.121,440.136,-120.251,176.447,37.700,157.184
C06986=1067.130,440.380,-120.300,176.457,37.713,157.187
C06987=1067.140,440.625,-120.350,176.466,37.726,157.191
C06988=1067.149,440.870,-120.398,176.476,37.740,157.195
C06989=1067.158,441.115,-120.447,176.485,37.753,157.199
C06990=1067.168,441.360,-120.496,176.494,37.767,157.202
C06991=1067.177,441.606,-120.545,176.504,37.781,157.206
C06992=1067.187,441.850,-120.594,176.514,37.794,157.210
C06993=1067.198,442.128,-120.650,176.525,37.810,157.214
C06994=1067.208,442.407,-120.706,176.536,37.826,157.218
C06995=1067.219,442.685,-120.762,176.547,37.841,157.223
C06996=1067.230,442.963,-120.818,176.558,37.857,157.227
C06997=1067.240,443.208,-120.867,176.568,37.871,157.231
C06998=1067.249,443.453,-120.917,176.578,37.885,157.235
C06999=1067.259,443.697,-120.966,176.587,37.899,157.239
C07000=1067.269,443.942,-121.016,176.597,37.913,157.242
C07001=1067.278,444.188,-121.065,176.608,37.927,157.246
C07002=1067.288,444.432,-121.115,176.618,37.941,157.250
C07003=1067.298,444.677,-121.164,176.628,37.955,157.254
C07004=1067.307,444.921,-121.214,176.638,37.969,157.258
C07005=1067.317,445.167,-121.264,176.648,37.984,157.262
C07006=1067.326,445.411,-121.314,176.658,37.998,157.266
C07007=1067.336,445.656,-121.363,176.668,38.012,157.270
C07008=1067.346,445.900,-121.414,176.679,38.027,157.274
C07009=1067.356,446.145,-121.464,176.689,38.041,157.278
C07010=1067.365,446.390,-121.514,176.700,38.056,157.282
C07011=1067.376,446.634,-121.564,176.710,38.070,157.287
C07012=1067.385,446.879,-121.614,176.721,38.085,157.291
C07013=1067.395,447.124,-121.664,176.731,38.100,157.295
C07014=1067.405,447.368,-121.715,176.741,38.114,157.299
C07015=1067.415,447.613,-121.764,176.752,38.129,157.303
C07016=1067.425,447.857,-121.815,176.763,38.144,157.307
C07017=1067.436,448.101,-121.865,176.774,38.159,157.311
C07018=1067.447,448.344,-121.914,176.784,38.173,157.315
C07019=1067.460,448.589,-121.962,176.795,38.187,157.319
C07020=1067.474,448.834,-122.011,176.805,38.200,157.323
C07021=1067.488,449.079,-122.058,176.815,38.213,157.327
C07022=1067.504,449.324,-122.104,176.825,38.226,157.331
C07023=1067.521,449.569,-122.150,176.835,38.239,157.334
C07024=1067.539,449.814,-122.195,176.845,38.251,157.338
C07025=1067.195,449.818,-122.455,176.834,38.382,157.373
C07026=1067.177,449.572,-122.411,176.825,38.370,157.369
C07027=1067.161,449.327,-122.365,176.815,38.358,157.366
C07028=1067.145,449.082,-122.318,176.805,38.345,157.362
C07029=1067.129,448.837,-122.270,176.794,38.332,157.359
C07030=1067.115,448.592,-122.223,176.784,38.318,157.355
C07031=1067.103,448.348,-122.174,176.772,38.304,157.351
C07032=1067.092,448.103,-122.125,176.762,38.290,157.347
C07033=1067.080,447.861,-122.075,176.750,38.276,157.342
C07034=1067.071,447.616,-122.025,176.740,38.260,157.338
C07035=1067.061,447.371,-121.975,176.729,38.246,157.334
C07036=1067.050,447.127,-121.925,176.719,38.231,157.330
C07037=1067.040,446.882,-121.874,176.709,38.217,157.326
C07038=1067.031,446.638,-121.824,176.697,38.202,157.322
C07039=1067.021,446.393,-121.774,176.687,38.188,157.318
C07040=1067.011,446.148,-121.724,176.677,38.173,157.314
C07041=1067.001,445.904,-121.674,176.666,38.159,157.309
C07042=1066.991,445.659,-121.624,176.656,38.144,157.305
C07043=1066.982,445.414,-121.574,176.646,38.130,157.301
C07044=1066.972,445.170,-121.525,176.635,38.116,157.297
C07045=1066.962,444.925,-121.474,176.625,38.102,157.293
C07046=1066.952,444.680,-121.424,176.615,38.088,157.289
C07047=1066.943,444.435,-121.375,176.605,38.073,157.285
C07048=1066.933,444.191,-121.325,176.595,38.059,157.281
C07049=1066.923,443.946,-121.275,176.584,38.045,157.278
C07050=1066.914,443.701,-121.225,176.574,38.031,157.274
C07051=1066.904,443.457,-121.176,176.564,38.017,157.270
C07052=1066.894,443.212,-121.126,176.554,38.003,157.266
C07053=1066.885,442.967,-121.078,176.544,37.989,157.262
C07054=1066.875,442.707,-121.025,176.534,37.974,157.258
C07055=1066.864,442.448,-120.973,176.524,37.960,157.254
C07056=1066.854,442.189,-120.920,176.512,37.946,157.250
C07057=1066.844,441.930,-120.869,176.502,37.931,157.246
C07058=1066.834,441.685,-120.820,176.492,37.918,157.242
C07059=1066.825,441.440,-120.770,176.483,37.904,157.238
C07060=1066.815,441.196,-120.721,176.473,37.890,157.234
C07061=1066.806,440.950,-120.672,176.464,37.877,157.231
C07062=1066.797,440.705,-120.623,176.455,37.864,157.227
C07063=1066.787,440.460,-120.574,176.445,37.850,157.223
C07064=1066.778,440.215,-120.526,176.435,37.837,157.220
C07065=1066.769,439.970,-120.477,176.426,37.823,157.216
C07066=1066.759,439.725,-120.428,176.416,37.810,157.212
C07067=1066.750,439.480,-120.379,176.406,37.797,157.209
C07068=1066.741,439.235,-120.331,176.398,37.783,157.205
C07069=1066.731,438.990,-120.282,176.388,37.771,157.202
C07070=1066.722,438.745,-120.233,176.379,37.757,157.198
C07071=1066.712,438.500,-120.185,176.370,37.745,157.195
C07072=1066.702,438.255,-120.136,176.361,37.731,157.191
C07073=1066.694,438.010,-120.088,176.351,37.718,157.187
C07074=1066.685,437.765,-120.040,176.342,37.706,157.184
C07075=1066.675,437.520,-119.991,176.333,37.693,157.180
C07076=1066.666,437.275,-119.944,176.324,37.680,157.177
C07077=1066.656,437.030,-119.895,176.315,37.667,157.173
C07078=1066.647,436.785,-119.847,176.306,37.654,157.170
C07079=1066.638,436.540,-119.799,176.296,37.641,157.166
C07080=1066.629,436.294,-119.751,176.288,37.629,157.163
C07081=1066.619,436.049,-119.703,176.278,37.616,157.160
C07082=1066.610,435.805,-119.655,176.270,37.604,157.156
C07083=1066.601,435.559,-119.607,176.261,37.591,157.153
C07084=1066.592,435.314,-119.560,176.252,37.579,157.149
C07085=1066.582,435.068,-119.512,176.243,37.566,157.146
C07086=1066.574,434.824,-119.464,176.235,37.554,157.143
C07087=1066.565,434.578,-119.416,176.226,37.541,157.139
C07088=1066.556,434.333,-119.369,176.217,37.529,157.136
C07089=1066.547,434.087,-119.321,176.208,37.517,157.133
C07090=1066.538,433.842,-119.273,176.200,37.504,157.130
C07091=1066.529,433.597,-119.226,176.192,37.492,157.126
C07092=1066.519,433.352,-119.178,176.182,37.480,157.123
C07093=1066.511,433.107,-119.131,176.174,37.468,157.120
C07094=1066.502,432.862,-119.083,176.165,37.455,157.116
C07095=1066.493,432.616,-119.036,176.157,37.444,157.113
C07096=1066.484,432.371,-118.989,176.149,37.432,157.110
C07097=1066.475,432.126,-118.941,176.140,37.419,157.107
C07098=1066.466,431.880,-118.894,176.132,37.407,157.104
C07099=1066.457,431.635,-118.847,176.123,37.395,157.100
C07100=1066.448,431.389,-118.800,176.115,37.383,157.097
C07101=1066.439,431.144,-118.752,176.106,37.372,157.094
C07102=1066.431,430.899,-118.706,176.098,37.360,157.091
C07103=1066.422,430.654,-118.658,176.090,37.348,157.088
C07104=1066.414,430.409,-118.612,176.082,37.336,157.085
C07105=1066.404,430.163,-118.565,176.073,37.324,157.081
C07106=1066.395,429.917,-118.518,176.065,37.313,157.078
C07107=1066.386,429.672,-118.471,176.057,37.301,157.075
C07108=1066.378,429.427,-118.424,176.049,37.289,157.072
C07109=1066.369,429.181,-118.377,176.041,37.278,157.069
C07110=1066.358,428.865,-118.317,176.031,37.263,157.065
C07111=1066.347,428.547,-118.257,176.020,37.248,157.061
C07112=1066.335,428.231,-118.197,176.009,37.233,157.057
C07113=1066.325,427.914,-118.137,176.000,37.219,157.054
C07114=1066.315,427.668,-118.091,175.992,37.207,157.051
C07115=1066.307,427.423,-118.045,175.984,37.196,157.048
C07116=1066.298,427.177,-117.998,175.976,37.185,157.045
C07117=1066.289,426.932,-117.952,175.968,37.173,157.042
C07118=1066.281,426.686,-117.906,175.961,37.162,157.039
C07119=1066.271,426.441,-117.860,175.953,37.151,157.036
C07120=1066.263,426.195,-117.813,175.945,37.140,157.033
C07121=1066.255,425.949,-117.767,175.937,37.129,157.030
C07122=1066.246,425.705,-117.721,175.929,37.118,157.027
C07123=1066.238,425.459,-117.675,175.922,37.107,157.024
C07124=1066.229,425.213,-117.630,175.914,37.096,157.022
C07125=1066.220,424.967,-117.583,175.906,37.085,157.019
C07126=1066.211,424.721,-117.537,175.898,37.074,157.016
C07127=1066.203,424.477,-117.491,175.891,37.063,157.013
C07128=1066.194,424.231,-117.446,175.883,37.052,157.010
C07129=1066.185,423.985,-117.400,175.875,37.041,157.007
C07130=1066.177,423.739,-117.354,175.868,37.030,157.004
C07131=1066.169,423.494,-117.309,175.861,37.020,157.002
C07132=1066.160,423.248,-117.262,175.853,37.009,156.999
C07133=1066.151,423.002,-117.217,175.846,36.998,156.996
C07134=1066.143,422.757,-117.171,175.838,36.987,156.993
C07135=1066.134,422.511,-117.126,175.831,36.977,156.991
C07136=1066.127,422.266,-117.080,175.823,36.966,156.988
C07137=1066.118,422.020,-117.035,175.816,36.956,156.985
C07138=1066.110,421.774,-116.989,175.809,36.945,156.982
C07139=1066.101,421.529,-116.944,175.801,36.934,156.980
C07140=1066.093,421.282,-116.899,175.794,36.924,156.977
C07141=1066.085,421.037,-116.853,175.786,36.913,156.974
C07142=1066.076,420.791,-116.808,175.780,36.903,156.972
C07143=1066.068,420.546,-116.763,175.772,36.893,156.969
C07144=1066.060,420.299,-116.718,175.765,36.882,156.966
C07145=1066.051,420.054,-116.673,175.758,36.872,156.964
C07146=1066.043,419.807,-116.628,175.751,36.861,156.961
C07147=1066.034,419.562,-116.583,175.743,36.851,156.958
C07148=1066.026,419.316,-116.538,175.736,36.841,156.956
C07149=1066.017,419.071,-116.493,175.729,36.831,156.953
C07150=1066.010,418.825,-116.448,175.722,36.821,156.951
C07151=1066.001,418.579,-116.403,175.715,36.810,156.948
C07152=1065.993,418.333,-116.358,175.708,36.800,156.945
C07153=1065.984,418.087,-116.314,175.701,36.790,156.943
C07154=1065.976,417.842,-116.269,175.694,36.780,156.940
C07155=1065.968,417.596,-116.224,175.687,36.770,156.938
C07156=1065.959,417.349,-116.180,175.680,36.760,156.935
C07157=1065.952,417.103,-116.135,175.673,36.750,156.933
C07158=1065.943,416.858,-116.090,175.666,36.740,156.930
C07159=1065.935,416.612,-116.045,175.660,36.730,156.928
C07160=1065.927,416.366,-116.001,175.653,36.720,156.925
C07161=1065.918,416.120,-115.956,175.645,36.710,156.922
C07162=1065.910,415.874,-115.912,175.639,36.701,156.920
C07163=1065.902,415.629,-115.868,175.632,36.690,156.918
C07164=1065.894,415.383,-115.823,175.625,36.681,156.915
C07165=1065.886,415.137,-115.779,175.618,36.671,156.913
C07166=1065.877,414.840,-115.725,175.610,36.659,156.910
C07167=1065.867,414.543,-115.672,175.603,36.647,156.907
C07168=1065.857,414.246,-115.619,175.594,36.636,156.904
C07169=1065.847,413.948,-115.565,175.586,36.624,156.901
C07170=1065.838,413.702,-115.521,175.579,36.614,156.898
C07171=1065.830,413.456,-115.477,175.573,36.605,156.896
C07172=1065.822,413.210,-115.433,175.566,36.596,156.894
C07173=1065.814,412.964,-115.389,175.559,36.586,156.891
C07174=1065.806,412.718,-115.346,175.553,36.577,156.889
C07175=1065.798,412.472,-115.302,175.546,36.567,156.886
C07176=1065.790,412.226,-115.258,175.540,36.558,156.884
C07177=1065.782,411.980,-115.214,175.533,36.548,156.882
C07178=1065.774,411.734,-115.170,175.527,36.539,156.880
C07179=1065.765,411.488,-115.127,175.521,36.530,156.877
C07180=1065.758,411.242,-115.083,175.513,36.520,156.875
C07181=1065.750,410.996,-115.039,175.507,36.511,156.872
C07182=1065.741,410.750,-114.996,175.501,36.502,156.870
C07183=1065.733,410.503,-114.952,175.494,36.493,156.868
C07184=1065.725,410.258,-114.908,175.488,36.483,156.866
C07185=1065.718,410.012,-114.864,175.481,36.474,156.863
C07186=1065.710,409.766,-114.821,175.475,36.465,156.861
C07187=1065.702,409.520,-114.778,175.469,36.456,156.859
C07188=1065.694,409.273,-114.734,175.462,36.447,156.857
C07189=1065.686,409.027,-114.691,175.456,36.438,156.854
C07190=1065.678,408.781,-114.647,175.450,36.428,156.852
C07191=1065.671,408.535,-114.604,175.443,36.419,156.850
C07192=1065.662,408.289,-114.561,175.437,36.410,156.847
C07193=1065.654,408.043,-114.518,175.431,36.401,156.845
C07194=1065.647,407.796,-114.474,175.425,36.392,156.843
C07195=1065.639,407.551,-114.431,175.419,36.383,156.841
C07196=1065.631,407.305,-114.388,175.413,36.374,156.839
C07197=1065.623,407.058,-114.344,175.407,36.365,156.836
C07198=1065.615,406.813,-114.301,175.401,36.357,156.834
C07199=1065.608,406.566,-114.258,175.394,36.347,156.832
C07200=1065.600,406.320,-114.215,175.388,36.339,156.830
C07201=1065.592,406.074,-114.172,175.382,36.330,156.828
C07202=1065.585,405.827,-114.129,175.376,36.321,156.825
C07203=1065.577,405.582,-114.087,175.369,36.312,156.823
C07204=1065.569,405.336,-114.043,175.364,36.303,156.821
C07205=1065.561,405.089,-114.001,175.358,36.295,156.819
C07206=1065.554,404.843,-113.957,175.352,36.286,156.817
C07207=1065.545,404.597,-113.915,175.345,36.277,156.815
C07208=1065.538,404.351,-113.872,175.339,36.269,156.813
C07209=1065.530,404.104,-113.830,175.334,36.260,156.811
C07210=1065.523,403.858,-113.788,175.328,36.252,156.808
C07211=1065.515,403.612,-113.744,175.322,36.243,156.806
C07212=1065.507,403.366,-113.702,175.316,36.234,156.804
C07213=1065.499,403.119,-113.660,175.309,36.226,156.802
C07214=1065.492,402.874,-113.616,175.304,36.217,156.800
C07215=1065.484,402.627,-113.574,175.298,36.209,156.798
C07216=1065.476,402.381,-113.532,175.292,36.200,156.796
C07217=1065.468,402.134,-113.490,175.286,36.192,156.794
C07218=1065.461,401.888,-113.447,175.281,36.183,156.792
C07219=1065.452,401.642,-113.404,175.275,36.175,156.790
C07220=1065.445,401.396,-113.362,175.269,36.167,156.788
C07221=1065.437,401.150,-113.320,175.262,36.159,156.786
C07222=1065.428,400.856,-113.270,175.256,36.148,156.783
C07223=1065.419,400.564,-113.220,175.249,36.139,156.781
C07224=1065.410,400.271,-113.170,175.243,36.129,156.779
C07225=1065.401,399.979,-113.120,175.235,36.119,156.776
C07226=1065.393,399.733,-113.078,175.230,36.111,156.774
C07227=1065.385,399.486,-113.036,175.224,36.103,156.772
C07228=1065.378,399.239,-112.994,175.218,36.094,156.770
C07229=1065.371,398.993,-112.952,175.213,36.086,156.768
C07230=1065.363,398.747,-112.910,175.207,36.078,156.766
C07231=1065.355,398.501,-112.868,175.201,36.070,156.764
C07232=1065.348,398.254,-112.826,175.196,36.061,156.762
C07233=1065.340,398.008,-112.784,175.190,36.053,156.760
C07234=1065.332,397.762,-112.742,175.185,36.046,156.759
C07235=1065.325,397.516,-112.701,175.179,36.038,156.757
C07236=1065.318,397.270,-112.659,175.173,36.029,156.755
C07237=1065.309,397.023,-112.617,175.168,36.021,156.753
C07238=1065.302,396.776,-112.576,175.162,36.014,156.751
C07239=1065.294,396.530,-112.534,175.157,36.005,156.749
C07240=1065.287,396.284,-112.493,175.151,35.998,156.747
C07241=1065.280,396.038,-112.451,175.145,35.990,156.745
C07242=1065.272,395.791,-112.409,175.140,35.982,156.743
C07243=1065.265,395.545,-112.368,175.134,35.974,156.741
C07244=1065.257,395.299,-112.326,175.129,35.966,156.740
C07245=1065.250,395.052,-112.285,175.123,35.958,156.738
C07246=1065.243,394.805,-112.244,175.118,35.950,156.736
